/// Initializes module
/// Remark: Aborts all ongoing transfers immediately
METHOD M_Init : BOOL
VAR_INPUT
END_VAR
eHandOverState := E_HandOverState.IDLE;
DeleteNextTransportData := FALSE;
RequestNextTransportData := FALSE;
HandoverComplete := FALSE;
FastSpeed := FALSE;

M_Init := TRUE;
END_METHOD

END_FUNCTION_BLOCK

// ---- 20_Product/10_BCF/11_Conv/12_E_Functions/10_Helper/FB_HandoverTracking.TcPOU

///Handover tracking while handing over the TU from the base tracking to next function
FUNCTION_BLOCK FB_HandoverTracking IMPLEMENTS I_HandoverListener
(**************************************************************************************
* Application : BoxControl Framework 
* Revision date : $Date: 2021-03-03 11:30:54 +0100 (ons, 03 mar 2021) $
* Author : CDC
* ------------------------------------------------------------------------------------ 
* © Swisslog AG 
* Swisslog is not liable for any usage of this source code that is not agreed 
* on between Swisslog and the other party. The mandatory legal liability remains 
* unaffected. 
* ------------------------------------------------------------------------------------ 
* Project revision history: 
* 
* 	VERSION 		DATE 			INITIALS 			DESCRIPTION 
* 	0.1 			22.08.2018 		herzig 				First implementation
*	0.2				05.10.2018		b7bolm				Review
* 
**************************************************************************************)
VAR_INPUT
	Param 						: ST_TransportControlParam; // Parameter of the transport control
	NextTransportData			: ST_TransportData; // Next transport data
	Enable						: BOOL; // Transport enable
	EnableHandOver 				: BOOL; // Transport enable handover
	OccupiedSensor				: BOOL; // Occupied PE, only to detect UFOs and data missmatch
	ZoneEndLength				: UINT; // Occupied position, distance from occupied to zone end
	TrackingLength				: UDINT; // Length of tracked distance
	MaxFrontEdgeDeviation		: UDINT := 100; // Max allowed deviation between occupied sensor and allocated zone
	DisableTU_Synchronisation	: BOOL; // Disable synchronisation of TU at occupied sensor
	DriveReady					: BOOL; // Drive is ready to be used
	DriveRunning				: BOOL; // Feedback drive is running
	EncoderValueInc				: UDINT; // Encoder value [inc]
	MaxEncoderValueInc			: UDINT; // Max encoder value [inc]
	RateIncPerMM				: LREAL; // Resolution number of increments for one mm
	iWindowTracking				: I_WindowTracking;  // Window tracking implementation
END_VAR
VAR_OUTPUT
	DriveRun					: BOOL; // Drive run
	DriveStop					: BOOL; // Stop drive
	FastSpeed					: BOOL; // Fast speed possible
	RequestNextTransportData 	: BOOL; // Request next transport data
	DeleteNextTransportData  	: BOOL; // Delete next transport data
	eHandOverState				: E_HandOverState; // Handover state
	eNextTakeOverState			: E_TakeOverState; // Takeover state of next position
	Initialized					: BOOL; // Module is initialized
	HandoverOngoing				: BOOL; // Handover ongoing, interface in interaction
	HandingOverTU				: BOOL; // Handing over the TU
END_VAR
VAR_IN_OUT
	ZoneData					: ST_ZoneData; // Zone data
	ErrorData 					: ST_ErrorDataSet; // Error data
END_VAR
VAR
	fbDebugMsg					: FB_DebugMsg; // Debug instance
	DebugMsg					: T_MAXSTRING; // Debug message
	TransportComplete			: BOOL; // Transport completed
	eTrackingState 				: E_HandoverTrackingState; // Handover state machine
	fbHandover					: FB_Handover; // Basic handover impementation
	TU_StartPosition			: UDINT; // TU start position
	TU_EndPosition				: UDINT; // TU end position
	TU_DetectedOnTracking 		: BOOL; // TU detected on tracking
	EndLengthEmpty 				: BOOL; // No TU in end length found
	TrackingZoneIndex 			: UINT; // Window tracking zone index
	TrackingUfoZoneIndex 		: UINT; // Window tracking zone index of ufo
	TrackingUfoReZoneIndex 		: UINT; // Window tracking zone index of ufo rear edge
	OccupiedZoneIndex 			: UINT; // Occupied zone index
	OccupiedTracking 			: BOOL; // Occupied tracking
	TransportEnable				: BOOL; // Transport hardstop
	TransportEnableHandOver		: BOOL; // Transport softstop, finish ongoing operations
	MonitorStoppingTU_Active	: BOOL; // Monitoring state is processed currently
	fbTrigOccupied				: R_TRIG; // Only check physical and tracking distance once
	fbZoneEndLengthClear		: FB_DisplacementMeter; // ZoneEndLenght clear
	DelayLength					: UDINT; // Delay length to clear conveyor end
	ZoneEndPosition				: UDINT; // End position of zone
END_VAR

//Input mapping
TransportEnable := Enable AND Param.rZoneEnable.Transport;
TransportEnableHandOver := EnableHandOver AND Param.rZoneEnable.HandOver AND Param.rExternalZoneEnable;

F_ResetError(Reset := FALSE, ErrorData := ErrorData);	

IF iWindowTracking = 0 OR
   TrackingLength = 0 THEN
	RETURN;
END_IF

// Initialization of the module
// Module initialization
IF NOT Initialized THEN
	RETURN;
END_IF

(**************************************************************************************************************
   Synchronization / Managing of physical TUs
***************************************************************************************************************)
// Always when a TU gets detected at sensor its checked if its synchronized to tracking.
// 1. If a TU gets detected and a corresponding tracked zone is found -> Everything fine
// 2. A TU gets detected without a tracked zone, try to find corresponding zone and align
// 3. TU can not be linked to a zone, add TU as new unknown zone to the tracking

// Remark: It is possible, that there is a small difference between zone and TU when the TU leaves
// the occupied sensor. 
IF NOT DisableTU_Synchronisation THEN
	fbTrigOccupied(CLK := OccupiedSensor);
	
	IF fbTrigOccupied.Q THEN
		OccupiedTracking := iWindowTracking.M_IsTU_Present(TrackingLength - ZoneEndLength);
	
		IF OccupiedTracking THEN
			// Sensor signal is corresponding to tracking zones
			;
		ELSE
			// Try to synchronize zone to occupied signal
			OccupiedZoneIndex := iWindowTracking.M_ResyncTU_FE(
									mAbsolutePosition 		:= TrackingLength - ZoneEndLength,
									mMaxFrontEdgeDeviation 	:= MaxFrontEdgeDeviation);
		
			// If physical TU could not be linked to a zone, handle as unidentified TU
			// Add it to tracking to follow normal handover procedure
			IF OccupiedZoneIndex = 0 THEN
				TrackingUfoZoneIndex := iWindowTracking.M_AddTU_FE(
											mTU_Index 			:= 0,
											mAbsolutePosition 	:= TrackingLength - ZoneEndLength,
											miActionListener 	:= 0);
											
				fbDebugMsg.M_SendInfoMsg(CONCAT('UFO front edge detected. Created ZoneIndex: ', UINT_TO_STRING(TrackingUfoZoneIndex)));	
			END_IF
		END_IF
		
	// Ufo found, wait for rear edge	
	ELSIF TrackingUfoZoneIndex > 0 AND NOT OccupiedSensor THEN
		TrackingUfoReZoneIndex := iWindowTracking.M_AddTU_RE(
									mAbsolutePosition 	:= TrackingLength - ZoneEndLength,
									mZoneIndex 			:= TrackingUfoZoneIndex);
									
		fbDebugMsg.M_SendInfoMsg(CONCAT('UFO rear edge detected. Completed ZoneIndex: ', UINT_TO_STRING(TrackingUfoReZoneIndex)));								
		TrackingUfoZoneIndex := 0;
	END_IF
END_IF

(**************************************************************************************************************
   Tracking state
***************************************************************************************************************)
MonitorStoppingTU_Active := FALSE;

CASE eTrackingState OF
	// Idle - Wait for a TU to handover
	E_HandoverTrackingState.WAITING_FOR_TU:	
		TrackingZoneIndex := 0;
		TransportComplete := FALSE;
		ZoneData.TransportControlData.TU_DataIndex := 0;
		ZoneData.TransportControlData.DataPresent := ZoneData.TransportControlData.TU_DataIndex > 0;
		
		// Check for a TU at occupation position (REMARK: Tracking zone begin != TU begin)
		TU_DetectedOnTracking := iWindowTracking.M_IsTU_Present(TrackingLength - ZoneEndLength);
 		
		// Scan for zones between occupation point and tracking end
		IF NOT EndLengthEmpty THEN	
			TrackingZoneIndex := iWindowTracking.M_GetLastZoneIndex(TrackingLength - ZoneEndLength , TrackingLength, TRUE);
			
			// A zone with TU present was found
			IF TrackingZoneIndex > 0 THEN
				// Get rear edge position of TU
				TU_EndPosition := iWindowTracking.M_GetTU_EndPosition(TrackingZoneIndex);
				// Check if TU already left conveyor
				IF TU_EndPosition > TrackingLength THEN
					// Get end position of zone
					ZoneEndPosition := iWindowTracking.M_GetZoneEndPosition(TrackingZoneIndex);
					
					// Search 2nd last zone, since TU of last zone already left conveyor
					IF ZoneEndPosition > (TrackingLength - ZoneEndLength) THEN
						TrackingZoneIndex := iWindowTracking.M_GetLastZoneIndex(TrackingLength - ZoneEndLength , ZoneEndPosition - 1, TRUE);
					ELSE
						// No zone found
						TrackingZoneIndex := 0;
					END_IF
				END_IF
				
				// A zone with a TU which is still on conveyor was found
				IF TrackingZoneIndex > 0 THEN 
					ZoneData.TransportControlData.TU_DataIndex := iWindowTracking.P_ZoneTable[TrackingZoneIndex].TU_Index;
					ZoneData.TransportControlData.DataPresent := ZoneData.TransportControlData.TU_DataIndex > 0;
					eTrackingState := E_HandoverTrackingState.MONITOR_STOPPING_TU;
				ELSE
					EndLengthEmpty := TRUE;
				END_IF
			ELSE
				EndLengthEmpty := TRUE;
			END_IF
			
		ELSIF TU_DetectedOnTracking  THEN
			// Get corresponding zone index
			TrackingZoneIndex := iWindowTracking.M_GetZoneIndex(TrackingLength - ZoneEndLength);
			EndLengthEmpty := FALSE;
			
			IF TrackingZoneIndex > 0 THEN
				ZoneData.TransportControlData.TU_DataIndex := iWindowTracking.P_ZoneTable[TrackingZoneIndex].TU_Index;
				ZoneData.TransportControlData.DataPresent := ZoneData.TransportControlData.TU_DataIndex > 0;
			END_IF
			
			eTrackingState := E_HandoverTrackingState.MONITOR_STOPPING_TU;
		END_IF
	
	// Handover is not initiated, ensure TU can stop properly
	E_HandoverTrackingState.MONITOR_STOPPING_TU:
		MonitorStoppingTU_Active := TRUE;
	
		IF TrackingZoneIndex > 0 THEN
			TU_StartPosition := iWindowTracking.M_GetTU_StartPosition(TrackingZoneIndex);
			
			// When zone is not in a valid range, forget index (> Occupation point)
			IF TU_StartPosition < (TrackingLength - ZoneEndLength) OR 
               NOT iWindowTracking.P_ZoneTable[TrackingZoneIndex].Used THEN
				TrackingZoneIndex := 0;
				DriveStop := FALSE;
				
				MonitorStoppingTU_Active := FALSE;
				eTrackingState := E_HandoverTrackingState.WAITING_FOR_TU;
				RETURN;
				
			// Check for overrun
			ELSIF TU_StartPosition > TrackingLength AND 
               iWindowTracking.P_ZoneTable[TrackingZoneIndex].TU_Index > 0 THEN
				// Overrun detected - Handover was not initated and TU could not stop on Tracking
				// Maybe condition to stop is wrong or available breaking distance is to short
				// Possible TU Index get deleted, because a crash could happen what maybe leads to 
				// Tu data inconsistency.
				iWindowTracking.P_ZoneTable[TrackingZoneIndex].TU_Index := 0;
				ZoneData.TransportControlData.TU_DataIndex := 0;
				ZoneData.TransportControlData.DataPresent := ZoneData.TransportControlData.TU_DataIndex > 0;
				fbDebugMsg.M_SendInfoMsg(CONCAT('Handover not initiated, TU_DataIndex deleted. ZoneIndex: ', UINT_TO_STRING(TrackingZoneIndex)));	
			END_IF
			
			// Wait until handover is initiated resp. ongoing
			IF fbHandover.eHandOverState = E_HandOverState.ACTIVE OR
			   fbHandover.eHandOverState = E_HandOverState.STOP OR
			   fbHandover.eHandOverState = E_HandOverState.INTERRUPTED OR 
               eNextTakeoverState = E_TakeOverState.ACTIVE THEN
			   
			   MonitorStoppingTU_Active := FALSE;
			   eTrackingState := E_HandoverTrackingState.MONITOR_HANDOVER_TU;
			END_IF
		ELSE
			MonitorStoppingTU_Active := FALSE;
			eTrackingState := E_HandoverTrackingState.WAITING_FOR_TU;
		END_IF
	
	// Handover was initiated, wait until TU left position
	E_HandoverTrackingState.MONITOR_HANDOVER_TU:
		IF TrackingZoneIndex > 0 THEN
			TU_StartPosition := iWindowTracking.M_GetTU_StartPosition(TrackingZoneIndex);
			TU_EndPosition := iWindowTracking.M_GetTU_EndPosition(TrackingZoneIndex);
			
			// Monitor zone if it is not in a valid range, forget index (> Occupation point)
			IF TU_StartPosition < (TrackingLength - ZoneEndLength) OR 
			   NOT iWindowTracking.P_ZoneTable[TrackingZoneIndex].Used THEN
				TrackingZoneIndex := 0;
				eTrackingState := E_HandoverTrackingState.WAITING_FOR_TU;
				RETURN;

			// Wait until transport is completed by
			// - Zone not available anymore
			// - Not occupied anymore
			// - Transport aborted or completed
			ELSIF NOT iWindowTracking.P_ZoneTable[TrackingZoneIndex].Used OR
			      NOT iWindowTracking.P_ZoneTable[TrackingZoneIndex].TU_Present OR
 			      fbHandover.eHandOverState = E_HandOverState.IDLE OR 
			      fbHandover.eHandOverState = E_HandOverState.UNDEFINED OR 
                  TransportComplete THEN		
				eTrackingState := E_HandoverTrackingState.WAITING_FOR_TU;
				
			// Monitor TU-DataIndex, and update it when it was deleted during handover
			ELSIF ZoneData.TransportControlData.TU_DataIndex <> iWindowTracking.P_ZoneTable[TrackingZoneIndex].TU_Index THEN
				iWindowTracking.P_ZoneTable[TrackingZoneIndex].TU_Index := ZoneData.TransportControlData.TU_DataIndex;
			END_IF
		ELSE
			eTrackingState := E_HandoverTrackingState.WAITING_FOR_TU;
		END_IF
// Default
ELSE
	eTrackingState := E_HandoverTrackingState.WAITING_FOR_TU;
END_CASE

(**************************************************************************************************************
   Handover state
***************************************************************************************************************)
// If an index was found between occupation point and tracking length
// Wait until TU left occupation point, to zone end length for handover
IF TrackingZoneIndex > 0 THEN 
	IF NOT fbZoneEndLengthClear.Run THEN
		TU_EndPosition := iWindowTracking.M_GetTU_EndPosition(TrackingZoneIndex);
		// TU rear edge is between occupied point and conveyor end
		IF (TrackingLength - ZoneEndLength) < TU_EndPosition AND TrackingLength >= TU_EndPosition THEN
			// Calculate distance from  TU rear edge to conveyor end 
			DelayLength := TrackingLength - TU_EndPosition;
		
			// Run zone end length clearing 
			fbZoneEndLengthClear(
				Run 				:= fbHandover.HandoverOngoing, 
				EncoderValueInc		:= EncoderValueInc,
				MaxEncoderValueInc 	:= MaxEncoderValueInc,
				RateIncPerMM		:= RateIncPerMM,
				SetPoint 			:= UDINT_TO_UINT(DelayLength));
		END_IF
	END_IF
END_IF

fbZoneEndLengthClear(
	EncoderValueInc		:= EncoderValueInc,
	MaxEncoderValueInc 	:= MaxEncoderValueInc,
	RateIncPerMM		:= RateIncPerMM);
	
fbHandover(
	Enable					:= TransportEnable AND
            				  (Param.rOperationState.eState = E_PositionState.STARTED OR
	        				   Param.rOperationState.eState = E_PositionState.STOPPING),
	RequestHandover			:= TrackingZoneIndex > 0 AND Param.rOperationState.eState = E_PositionState.STARTED AND TransportEnableHandOver,
	NextZonePresent			:= Param.reNextFunctionNumber > 0,
	HandoverComplete		:= fbZoneEndLengthClear.Q,
	DriveReady				:= DriveReady,
	iListener				:= THIS^,
	FastSpeed				=> FastSpeed,
	DriveRun				=> DriveRun,
	eHandOverState			=> eHandOverState,
	eNextTakeOverState		=> eNextTakeOverState,
	RequestNextTransportData=> RequestNextTransportData,
	DeleteNextTransportData	=> DeleteNextTransportData,
	HandoverOngoing			=> HandoverOngoing,
	NextTransportData		:= NextTransportData,
	ErrorData				:= ErrorData);

IF fbZoneEndLengthClear.Q THEN
	fbZoneEndLengthClear(RUN := FALSE);
END_IF

ZoneData.TransportControlData.eHandOverState := eHandOverState;
ZoneData.TransportControlData.DataPresent := ZoneData.TransportControlData.TU_DataIndex <> 0;
ZoneData.TransportControlData.SensorOccupied := iWindowTracking.M_IsTU_Present(TrackingLength - ZoneEndLength);
ZoneData.TransportControlData.TU_LeadingEdgePos := 0;

DriveStop := (fbHandover.HandoverOngoing AND NOT fbHandover.DriveRun AND NOT fbHandover.DriveRequest) OR 
             (NOT fbHandover.HandoverOngoing AND MonitorStoppingTU_Active AND
			  (eHandOverState <> E_HandoverState.READY OR eNextTakeOverState <> E_TakeOverState.READY));

HandingOverTU := fbHandOver.HandoverOngoing;

/// Handover completed event
METHOD M_HandoverCompleteEvent

IF eTrackingState = E_HandoverTrackingState.MONITOR_HANDOVER_TU THEN
	TransportComplete := TRUE;
	
	IF iWindowTracking <> 0 THEN
		IF TrackingZoneIndex > 0 THEN
			iWindowTracking.M_DeleteZone(mZoneIndex := TrackingZoneIndex);
		END_IF
	END_IF
END_IF
END_METHOD

METHOD M_HandoverStartEvent
END_METHOD

/// Initialize module
METHOD M_Init : BOOL
VAR_INPUT
END_VAR
fbHandover.M_Init();

eTrackingState := E_HandoverTrackingState.WAITING_FOR_TU;
Initialized := TRUE;
M_Init := TRUE;
END_METHOD

END_FUNCTION_BLOCK

// ---- 20_Product/30_Toolbox/17_WindowTracking/10_Core/FB_DisplacementMeter.TcPOU
FUNCTION_BLOCK FB_DisplacementMeter
(**************************************************************************************
 * 	Application		:	BoxControl Framework
 *	Revision		:	$Revision: 354283 $
 *	Revision date	:	$Date: 2015-09-02 11:51:42 +0200 (Mi, 02 Sep 2015) $
 *	Last changed by	:	$Author: d7mangc $
 *	URL				:	$URL: http://almscdc.swisslog.com/repo/SWPD/Development/BoxControlFramework/20_Release/trunk/01_Software/BoxControlFramework/BoxControlFramework/JumpStart/11_Library/10_Application/10_Base/13_TimerCounter/FB_Timer.TcPOU $
 *
 *	Purpose			:	Measures displacement based on encoder value. Output Q gets true when setpoint is reached
 *						
 *
 * ------------------------------------------------------------------------------------
 *	Copyright Swisslog [IP AG], Switzerland. All rights reserved.
 * 
 * ------------------------------------------------------------------------------------
 *	
 * 	Revision History: 
 *
 * 	VERSION			DATE			INITIALS			DESCRIPTION
 *	0.1				01.01.2001		swl					Example
 *
 **************************************************************************************)
VAR_INPUT
	Run             	: BOOL; // Start process on rising edge
	EncoderValueInc		: UDINT; // Encoder value [inc], Ascending = forward
	MaxEncoderValueInc	: UDINT; // Max encoder value [inc]
	RateIncPerMM		: LREAL; // Ratio - How many increments represent one mm
	SetPoint			: DINT; // Displacement value where Q is set true (negative: backward direction, positive: forward direction)
	StartPoint		    : DINT; // Starting position (offset) for displacement measurement [mm] (negative : backward direction, positive: forward direction)
END_VAR
VAR_OUTPUT
	Q		 			: BOOL; // True when setpoint reached
	DisplacementInc		: DINT; // Current displacement [inc] (negative : backward direction, positive: forward direction)
	Displacement		: DINT; // Current displacement [mm] (negative : backward direction, positive: forward direction)
END_VAR
VAR
	Trg			     	: BOOL; // Trigger detection for start signal
	LastEncoderValueInc	: UDINT; // Last encoder value [inc]
	Inc 			 	: DINT; // increments
END_VAR

IF Run THEN
	// Detect start trigger and preset values
	IF NOT Trg AND Run THEN
		LastEncoderValueInc := EncoderValueInc;
		DisplacementInc := LREAL_TO_DINT(DINT_TO_LREAL(StartPoint) * RateIncPerMM);
		Displacement := 0;
	END_IF

	Inc := UDINT_TO_DINT(EncoderValueInc) - UDINT_TO_DINT(LastEncoderValueInc);
	IF ABS(Inc) > UDINT_TO_DINT(MaxEncoderValueInc/2) THEN
		IF Inc < 0 THEN
			Inc := Inc + 1 + UDINT_TO_DINT(MaxEncoderValueInc);
		ELSE
			Inc := UDINT_TO_DINT(EncoderValueInc) - (UDINT_TO_DINT(LastEncoderValueInc) + UDINT_TO_DINT(MaxEncoderValueInc)) - 1;
		END_IF
	END_IF
	
	// Update last encoder value
	LastEncoderValueInc := EncoderValueInc;
	
	// Update outputs
	IF NOT Q THEN
		DisplacementInc := DisplacementInc + Inc;
		
		IF RateIncPerMM > 0 THEN
			Displacement := LREAL_TO_DINT(DINT_TO_LREAL(DisplacementInc) / RateIncPerMM);
		ELSE
			Displacement := 0;
		END_IF
		
		// To ensure counting direction is as desired,
		// decision is based on the sign of setpoint
		IF SetPoint >= 0 THEN
			IF Displacement >= SetPoint THEN
				Q := TRUE;
			END_IF
		ELSE
			IF Displacement <= SetPoint THEN
				Q := TRUE;
			END_IF
		END_IF
	END_IF
ELSE
	// Reset outputs
	Q := FALSE;
END_IF

Trg := Run;

END_FUNCTION_BLOCK

// ---- 20_Product/10_BCF/11_Conv/12_E_Functions/10_Helper/FB_HandoverTrackingDivert.TcPOU
/// Functionality to control a handover process from a tracking conveyor
FUNCTION_BLOCK FB_HandoverTrackingDivert IMPLEMENTS I_HandoverListener
(************************************************************************************** 
* 	Application 		: BoxControl Framework 
* 	Revision 			: $Revision: 408723 $ 
* 	Revision date 		: $Date: 2018-06-27 13:49:08 +0200 (Wed, 27 Jun 2018) $ 
* 	Last changed by 	: $Author: b7bolm $ 
* 	URL 				: $URL: http://almscdc.swisslog.com/repo/SWPD/Development/BoxControlFramework/21_Projects/BCF_2.0/trunk/BCF/BCF/JumpStart/20_Product/10_App/12_E_Functions/10_Lib/10_Conv/FB_FunctionList.TcPOU $ 
* ------------------------------------------------------------------------------------ 
* 	© Swisslog AG 
* 	Swisslog is not liable for any usage of this source code that is not agreed 
* 	on between Swisslog and the other party. The mandatory legal liability remains 
* 	unaffected. 
* ------------------------------------------------------------------------------------ 
* 	Revision History: 
* 
* 	VERSION 		DATE 			INITIALS 			DESCRIPTION 
* 	0.1 			22.08.2018 		herzig 				First implementation
*	0.2				05.10.2018		b7bolm				Review
* 
**************************************************************************************)
VAR_INPUT
	Param 						: ST_TransportControlParam; // Parameter of the transport control
	NextTransportData			: ST_TransportData; // Next transport data
	Enable						: BOOL; // Transport enable
	EnableHandOver 				: BOOL; // Transport enable handover
	DivertPosition				: UDINT; // Merging position on tracking
	DivertingTolerance			: UDINT; // Merging tolerance to allow merging
	DivertRearEdge				: BOOL; // Divert on rear edge of TU
	DriveDelayDistance			: DINT;  // Distance to drive until position is free
	DriveReady					: BOOL; // Drive is ready to be used
	EncoderValueInc				: UDINT; // Encoder value [inc]
	MaxEncoderValueInc			: UDINT; // Max encoder value [inc]
	RateIncPerMM				: LREAL; // Resolution amount of increment per mm
	iWindowTracking				: I_WindowTracking;  // Window tracking implementation
END_VAR

VAR_OUTPUT
	DriveRun					: BOOL; // Drive run
	DriveStop					: BOOL; // Stop drive
	FastSpeed					: BOOL; // Fast speed possible
	RequestNextTransportData 	: BOOL; // Request next transport data
	DeleteNextTransportData  	: BOOL; // Delete next transport data
	eHandOverState				: E_HandOverState; // Handover state
	eNextTakeOverState			: E_TakeOverState; // Takeover state of next position
	Initialized					: BOOL; // Module is initialized
	AvailableZoneIndex			: UINT; // Current valid zone index
	HandoverOngoing				: BOOL; // Handover ongoing, interface in interaction
END_VAR

VAR_IN_OUT
	ZoneData					: ST_ZoneData; // Zone data
	ErrorData 					: ST_ErrorDataSet; // Error data
END_VAR

VAR
	fbDebugMsg					: FB_DebugMsg; // Debug instance
	DebugMsg					: T_MAXSTRING; // Debug message
	fbHandover					: FB_Handover; // Basic handover impementation
	DistanceToTU				: DINT; // Distance to TU from diverting point
	TransportEnable				: BOOL; // Transport hardstop
	TransportEnableHandOver		: BOOL; // Transport softstop, finish ongoing operations
	TU_IndexOfZone				: DINT; // TU index of tracking zone
	TrackingZoneIndex 			: UINT; // Tracking zone index
	fbZoneEndLengthClear		: FB_DisplacementMeter; // ZoneEndLenght clear
END_VAR

//Input mapping
TransportEnable := Enable AND Param.rZoneEnable.Transport;
TransportEnableHandOver := EnableHandOver AND Param.rZoneEnable.HandOver AND Param.rExternalZoneEnable;

F_ResetError(Reset := FALSE, ErrorData := ErrorData);	

IF iWindowTracking = 0 THEN
	RETURN;
END_IF

// Initialization of the module
// Module initialization
IF NOT Initialized THEN
	RETURN;
END_IF

(**************************************************************************************************************
   Determine zone for this position
***************************************************************************************************************)
AvailableZoneIndex := 0;
TU_IndexOfZone := 0;
ZoneData.TransportControlData.DataPresent := FALSE;
ZoneData.TransportControlData.TU_DataIndex := 0;

// Wait until a zone can be found at divert point
IF TrackingZoneIndex = 0 THEN
	IF DivertRearEdge THEN
		TrackingZoneIndex := iWindowTracking.M_GetFirstZoneIndex(DivertPosition, DivertPosition + DivertingTolerance, TRUE);
	ELSE
		TrackingZoneIndex := iWindowTracking.M_GetZoneIndex(DivertPosition);	
	END_IF
END_IF

// When a possible zone was found, validate and monitor it
IF TrackingZoneIndex > 0 THEN
	// As long the zone is valid
	IF iWindowTracking.P_ZoneTable[TrackingZoneIndex].Used THEN
		// Divert on rear edge
		IF DivertRearEdge THEN
			// Zone gets monitored as long it is in a certain range 
			DistanceToTU := iWindowTracking.M_GetDistanceToTU_End(DivertPosition, TrackingZoneIndex);
		ELSE
			// Zone gets monitored as long it is in a certain range 
			DistanceToTU := iWindowTracking.M_GetDistanceToTU_Start(DivertPosition, TrackingZoneIndex);
		END_IF
		
		// TU needs to pass divert point and stays available for distance (Divertingtolerance)
		IF DistanceToTU <= 0 AND ABS(DistanceToTU) <= UDINT_TO_DINT(DivertingTolerance) THEN
			// When position is occupied, its a possible next for this position
			IF iWindowTracking.P_ZoneTable[TrackingZoneIndex].TU_Present THEN			
				TU_IndexOfZone := iWindowTracking.P_ZoneTable[TrackingZoneIndex].TU_Index;
			
				ZoneData.TransportControlData.DataPresent := TU_IndexOfZone <> 0;
				ZoneData.TransportControlData.TU_DataIndex := TU_IndexOfZone;
				
				AvailableZoneIndex := TrackingZoneIndex;	
			END_IF
			
		// TU left divert tolerance range
		ELSIF DistanceToTU <= 0 AND ABS(DistanceToTU) > UDINT_TO_DINT(DivertingTolerance) THEN
			TrackingZoneIndex := 0;
		END_IF
	END_IF
END_IF

(**************************************************************************************************************
   Handover state
***************************************************************************************************************)
// Delay after enabling handover, set as soon transport gets started
fbZoneEndLengthClear(
	EncoderValueInc		:= EncoderValueInc,
	MaxEncoderValueInc 	:= MaxEncoderValueInc,
	RateIncPerMM		:= RateIncPerMM);
	
fbHandover(
	Enable					:= TransportEnable AND
            				  (Param.rOperationState.eState = E_PositionState.STARTED OR
	         				   Param.rOperationState.eState = E_PositionState.STOPPING),
	RequestHandover			:= AvailableZoneIndex > 0 AND Param.rOperationState.eState = E_PositionState.STARTED AND TransportEnableHandOver,
	NextZonePresent			:= Param.reNextFunctionNumber > 0,
	HandoverComplete		:= fbZoneEndLengthClear.Q,
	DriveReady				:= DriveReady,
	iListener				:= THIS^,
	FastSpeed				=> FastSpeed,
	DriveRun				=> DriveRun,
	eHandOverState			=> eHandOverState,
	eNextTakeOverState		=> eNextTakeOverState,
	RequestNextTransportData=> RequestNextTransportData,
	DeleteNextTransportData	=> DeleteNextTransportData,
	HandoverOngoing			=> HandoverOngoing,
	NextTransportData		:= NextTransportData,
	ErrorData				:= ErrorData);
	
IF fbZoneEndLengthClear.Q THEN
	fbZoneEndLengthClear(RUN := FALSE);
END_IF
	
ZoneData.TransportControlData.eHandOverState := eHandOverState;
ZoneData.TransportControlData.DataPresent := ZoneData.TransportControlData.TU_DataIndex <> 0;
ZoneData.TransportControlData.SensorOccupied := AvailableZoneIndex > 0;
ZoneData.TransportControlData.Occupied := AvailableZoneIndex > 0;
ZoneData.TransportControlData.TU_LeadingEdgePos := 0;

DriveStop := (fbHandover.HandoverOngoing AND NOT fbHandover.DriveRun AND NOT fbHandover.DriveRequest);

/// Handover completed event
METHOD M_HandoverCompleteEvent
TrackingZoneIndex := 0;
END_METHOD

/// Handover initiated -> Active
METHOD M_HandoverStartEvent
VAR
	mZoneDeleted	: BOOL;
END_VAR

IF AvailableZoneIndex > 0 THEN
	IF iWindowTracking <> 0 THEN
		mZoneDeleted := iWindowTracking.M_DeleteZone(AvailableZoneIndex);
		IF mZoneDeleted THEN
			DebugMsg := CONCAT('Zone deleted from tracking by divert. ZoneIndex: ', UINT_TO_STRING(AvailableZoneIndex));
			
		ELSE
			DebugMsg := CONCAT('Zone delete from tracking by divert not possible. ZoneIndex: ', UINT_TO_STRING(AvailableZoneIndex));
		END_IF
		fbDebugMsg.M_SendInfoMsg(DebugMsg);
	END_IF
	
	// Run zone end length clearing 
	fbZoneEndLengthClear(
		Run 				:= TRUE, 
		EncoderValueInc		:= EncoderValueInc,
		MaxEncoderValueInc 	:= MaxEncoderValueInc,
		RateIncPerMM 		:= RateIncPerMM,
		SetPoint 			:= DriveDelayDistance);
END_IF
END_METHOD

/// Initialize module
METHOD M_Init : BOOL
VAR_INPUT
END_VAR
fbHandover.M_Init();

Initialized := TRUE;
M_Init := TRUE;
END_METHOD

END_FUNCTION_BLOCK

// ---- 20_Product/10_BCF/11_Conv/12_E_Functions/10_Helper/FB_SpeedControl.TcPOU
FUNCTION_BLOCK FB_SpeedControl
(**************************************************************************************
 * 	Application		:	BoxControl Framework
 *	Revision		:	$Revision: 404529 $
 *	Revision date	:	$Date: 2018-04-23 08:21:38 +0200 (Mo., 23 Apr 2018) $
 *	Last changed by	:	$Author: b7bolm $
 *	URL				:	$URL: http://almscdc.swisslog.com/repo/SWPD/Development/BoxControlFramework/20_Release/trunk/01_Software/BCF/BCF/JumpStart/20_Product/10_App/12_E_Functions/10_Lib/10_Conv/10_Functions/FB_SpeedControl.TcPOU $
 *
 *	Purpose			:	Speed control
 *
 * ------------------------------------------------------------------------------------
 *	Copyright Swisslog [IP AG], Switzerland. All rights reserved.
 * 
 * ------------------------------------------------------------------------------------
 *	
 * 	Revision History: 
 *
 * 	VERSION			DATE			INITIALS			DESCRIPTION
 *	0.1				01.01.2001		swl					Example
 *
 **************************************************************************************)
VAR_INPUT
	FastSpeed 		: BOOL; // Fast speed
	SetSpeed 		: REAL; // Set speed of the zone [m/s]
	SpeedSlow 		: INT;  // Speed slow [%]
	SpeedFast 		: INT;  // Speed fast [%]
END_VAR

VAR
	MasterSpeed		: INT; // Master speed [%]
END_VAR

VAR_OUTPUT
	CommandSpeed 	: INT; // Command speed [mm/s]
END_VAR

// Get Master speed from subsystem
IF __ISVALIDREF(SubsystemRegistry.rSubsystemInterface) THEN
	MasterSpeed := SubsystemRegistry.rSubsystemInterface.Out.MasterSpeed;
ELSE
	MasterSpeed := 100;
END_IF

// Calculate command speed
IF FastSpeed THEN
	CommandSpeed := REAL_TO_INT(SetSpeed * 1000 * SpeedFast / 100 * MasterSpeed / 100);
ELSE
	CommandSpeed := REAL_TO_INT(SetSpeed * 1000 * SpeedSlow / 100 * MasterSpeed / 100);
END_IF

END_FUNCTION_BLOCK

// ---- 20_Product/10_BCF/11_Conv/12_E_Functions/10_Helper/FB_SpeedControlRamp.TcPOU
FUNCTION_BLOCK FB_SpeedControlRamp
(**************************************************************************************
 * 	Application		:	BoxControl Framework
 *	Revision		:	$Revision: 404529 $
 *	Revision date	:	$Date: 2018-04-23 08:21:38 +0200 (Mo., 23 Apr 2018) $
 *	Last changed by	:	$Author: b7bolm $
 *	URL				:	$URL: http://almscdc.swisslog.com/repo/SWPD/Development/BoxControlFramework/20_Release/trunk/01_Software/BCF/BCF/JumpStart/20_Product/10_App/12_E_Functions/10_Lib/10_Conv/10_Functions/FB_SpeedControl.TcPOU $
 *
 *	Purpose			:	Speed control with acceleration/deceleration ramps
 *
 * ------------------------------------------------------------------------------------
 *	Copyright Swisslog [IP AG], Switzerland. All rights reserved.
 * 
 * ------------------------------------------------------------------------------------
 *	
 * 	Revision History: 
 *
 * 	VERSION			DATE			INITIALS			DESCRIPTION
 *	0.1				01.01.2001		swl					Example
 *
 **************************************************************************************)
VAR_INPUT
	DriveRun 				: BOOL; // Drive run
	TU_InBrakingZone 		: BOOL; // TU is within the braking zone 
	SetSpeed 				: REAL; // Set speed of the zone [m/s]
	SpeedSlow 				: INT; // Speed slow [%]
	SpeedFast 				: INT; // Speed fast [%]
	Acceleration   	 		: INT; // Accelaration [mm/s^2]
	Deceleration   	 		: INT; // Deceleration [mm/s^2]
	TransportControlData 	: ST_TransportControlData;
	SpeedPrevZone			: INT; // Speed from previous zone
	MinimumSpeed			: INT; // Minimum speed [mm/s]
END_VAR
VAR
	MasterSpeed				: INT; // Master speed [%]
	fbGetCurTaskIdx  		: GETCURTASKINDEX;
	CycleTime       		: REAL; // System cycletime [s]
	DesiredSpeed 			: INT; // Desired speed [mm/s]
	State 					: E_SpeedControlState; // Speed control state
	SpeedDelta				: INT; // Speed delta [mm/s]
END_VAR
VAR_OUTPUT
	CommandSpeed 			: INT; // Command speed [mm/s]
END_VAR

// Get current cycle time
fbGetCurTaskIdx();
CycleTime := UDINT_TO_REAL(_TaskInfo[fbGetCurTaskIdx.index].CycleTime) / 10000000;

// Get Master speed from subsystem
IF __ISVALIDREF(SubsystemRegistry.rSubsystemInterface) THEN
	MasterSpeed := SubsystemRegistry.rSubsystemInterface.Out.MasterSpeed;
ELSE
	MasterSpeed := 100;
END_IF


(**********************************************************************************************************
   Calculate desired speed
***********************************************************************************************************)
// When TakeOver starts sync CommandSpeed with previous zone
IF TransportControlData.eTakeOverState = E_TakeOverState.READY AND
   TransportControlData.eTransportState <> E_TransportState.MULTI_TU THEN
	CommandSpeed := SpeedPrevZone;
	
// In TakeOver sync desired speed with previous zone
ELSIF TransportControlData.eTransportState = E_TransportState.TAKEOVER AND NOT TU_InBrakingZone THEN
	DesiredSpeed := SpeedPrevZone;

// Check if fast speed is active then run at fast speed	
ELSIF TransportControlData.FastSpeedActive THEN
	DesiredSpeed := REAL_TO_INT(SetSpeed * 1000 * SpeedFast / 100 * MasterSpeed / 100);
	
// When not in braking zone run at low speed
ELSIF NOT TU_InBrakingZone THEN
	DesiredSpeed := REAL_TO_INT(SetSpeed * 1000 * SpeedSlow / 100 * MasterSpeed / 100);
	
// If not in TakeOver, Fast speed and TU is in braking zone request for minimum speed
ELSE
	DesiredSpeed := MinimumSpeed;
END_IF

// Limit the desired speed between system MinimumSpeed and the zone SetSpeed
IF DriveRun THEN
	DesiredSpeed := LIMIT(MinimumSpeed, DesiredSpeed, REAL_TO_INT(SetSpeed * 1000.0));	
END_IF


(**********************************************************************************************************
   Speed control state
***********************************************************************************************************)
CASE State OF
	
// STOPPED
	E_SpeedControlState.STOPPED:
		DesiredSpeed := 0;
		CommandSpeed := 0;
		// Wait for run command  
		IF DriveRun THEN
			State := E_SpeedControlState.Accelerate;
		END_IF
		
// ACCELERATE
	E_SpeedControlState.ACCELERATE:
		IF NOT DriveRun THEN
			State := E_SpeedControlState.Stopped;
			
		ELSIF CommandSpeed >= DesiredSpeed THEN
		 	State := E_SpeedControlState.Running;
		ELSE
			// Cyclic delta in speed [mm/s / cycle]
			SpeedDelta := REAL_TO_INT(Acceleration * CycleTime);
			CommandSpeed := LIMIT(MinimumSpeed, CommandSpeed + SpeedDelta, REAL_TO_INT(SetSpeed * 1000.0));
		END_IF
		
// RUNNING	
	E_SpeedControlState.RUNNING:
		IF NOT DriveRun THEN
			State := E_SpeedControlState.Stopped;
			
		ELSIF CommandSpeed > DesiredSpeed THEN
			State := E_SpeedControlState.Decelerate;
			
		ELSIF CommandSpeed < DesiredSpeed THEN
			State := E_SpeedControlState.Accelerate;
		END_IF
	
// DECELERATE	
	E_SpeedControlState.DECELERATE:
		IF NOT DriveRun THEN
			State := E_SpeedControlState.Stopped;
			
		ELSIF CommandSpeed < DesiredSpeed THEN
			State := E_SpeedControlState.Accelerate;		
		ELSE
			// Cyclic delta in speed [mm/s / cycle]
			SpeedDelta := REAL_TO_INT(Deceleration * CycleTime);
			CommandSpeed := LIMIT(MinimumSpeed, CommandSpeed - SpeedDelta, REAL_TO_INT(SetSpeed * 1000.0));
		END_IF
	
ELSE
	State := E_SpeedControlState.STOPPED;
END_CASE

END_FUNCTION_BLOCK

// ---- 20_Product/10_BCF/11_Conv/12_E_Functions/10_Helper/FB_Takeover.TcPOU
/// Basic takeover implementation to satisfy interface
FUNCTION_BLOCK FB_Takeover
(**************************************************************************************
* Application : BoxControl Framework 
* Revision date : $Date: 2021-04-01 10:33:04 +0200 (tor, 01 apr 2021) $
* Author : CDC
* ------------------------------------------------------------------------------------ 
* © Swisslog AG 
* Swisslog is not liable for any usage of this source code that is not agreed 
* on between Swisslog and the other party. The mandatory legal liability remains 
* unaffected. 
* ------------------------------------------------------------------------------------ 
* Project revision history: 
* 
* VERSION 	DATE 		INITIALS 	DESCRIPTION 
* 	VERSION 		DATE 			INITIALS 			DESCRIPTION 
* 	0.1 			22.08.2018 		herzig 				First implementation
*	0.2				05.10.2018		b7bolm				Review
* 
**************************************************************************************)

VAR_INPUT
	Enable						: BOOL; // Allow handover in general  
	RequestTakeover				: BOOL; // Rising edge initiates a new transport
	AbortTakeover				: BOOL; // Takeover must be aborted
	PrevZonePresent 			: BOOL;	 // Previous zone is known
	EncoderValue				: UDINT; // Encoder signal of movement
	MaxEncoderValue 			: UDINT; // Maximum encoder signal
	EncoderRate					: LREAL; // Rate from encoder to mm signal
	DriveReady					: BOOL; // Drive is ready to be used
	iListener 					: I_TakeoverListener; // Listener for any takeover events
END_VAR
VAR_OUTPUT
	DriveRun					: BOOL; // Switch on drive
	DriveRequest				: BOOL; // Request to get drive ready
	eTakeOverState				: E_TakeOverState; // Takeover state
	ePrevHandOverState			: E_HandOverState; // Handoverstate of previous zone
	RequestPrevTransportData 	: BOOL; // Request previous transport data
	DeletePrevTransportData 	: BOOL; // Delete previous transport dat
	TakeoverOngoing				: BOOL; // A takeover is ongoing, statemachine in operation
END_VAR
VAR_IN_OUT
	PrevTransportData			: ST_TransportData; // Next transport data
	ErrorData					: ST_ErrorDataSet; // Error slot
END_VAR
VAR
	TU_Index					: DINT; // TU index
	fbDebugMsg					: FB_DebugMsg; // Debug instance
	DebugMsg					: T_MAXSTRING; // Debug message
END_VAR


F_ResetError(Reset := FALSE, ErrorData := ErrorData);	

(*************************************************************************
  Undefined
*************************************************************************)
CASE eTakeOverState OF
	// Undefined
	E_TakeOverState.UNDEFINED:
		TakeoverOngoing := FALSE;
		eTakeOverState := E_TakeOverState.IDLE;


(*************************************************************************
  Idle
*************************************************************************)
	E_TakeOverState.IDLE:
		TakeoverOngoing := FALSE;
		DeletePrevTransportData := FALSE;
		RequestPrevTransportData := NOT PrevZonePresent;
		DriveRequest := FALSE;
		DriveRun := FALSE;
		
		IF RequestTakeover THEN
			// If the zone is internally ready for takeover
			IF Enable  AND
			   ErrorData.ErrorType <> E_ErrorType.ERROR THEN
				  
				// If prev zone or function is available
				IF PrevZonePresent THEN
					IF PrevTransportData.rTransportControlData.eHandOverState = E_HandOverState.READY THEN
						DriveRequest := TRUE;
						
						IF DriveReady THEN
							eTakeOverState := E_TakeOverState.READY;
						END_IF
					END_IF
				END_IF
			END_IF
		END_IF


(*************************************************************************
  Ready
*************************************************************************)
	E_TakeOverState.READY:
		TakeoverOngoing := FALSE;

		IF NOT Enable OR NOT RequestTakeover OR
		   ErrorData.ErrorType = E_ErrorType.ERROR OR
           NOT PrevZonePresent OR
           NOT DriveReady THEN  
			eTakeOverState := E_TakeOverState.IDLE;

		// Previous position is ready to handover
		ELSIF PrevTransportData.rTransportControlData.eHandOverState = E_HandOverState.READY THEN
			// Set drive on to create minimum TU gap
			DriveRun := TRUE;
			
			IF iListener <> 0 THEN
			   iListener.M_TakeoverStartEvent();
		   	END_IF

			// Move TU-data index from previous to own zone
			TU_Index := F_MoveTU_DataIndex(
								eFunctionNumber := PrevTransportData.eFunctionNumber,
								mZoneNumber 	:= PrevTransportData.ZoneNumber);

			IF iListener <> 0 THEN
				iListener.M_TU_IndexMovedEvent(TU_Index);
			END_IF

			eTakeOverState := E_TakeOverState.ACTIVE;
		END_IF


(*************************************************************************
  Active
*************************************************************************)
	E_TakeOverState.ACTIVE:
		DriveRun := TRUE;
		DriveRequest := FALSE;
		
		// Interrupt takeover if previous position stopped handover
		IF PrevTransportData.rTransportControlData.eHandOverState = E_HandOverState.STOP THEN
			DriveRun := FALSE;
			eTakeOverState := E_TakeOverState.INTERRUPTED;

		// Stop takeover from own cause
		ELSIF NOT Enable OR NOT DriveReady OR ErrorData.ErrorType = E_ErrorType.ERROR THEN	  
			DriveRun := FALSE;
			eTakeOverState := E_TakeOverState.STOP;
			
			IF iListener <> 0 THEN
			   iListener.M_TakeoverStopEvent();
		   	END_IF

		// Regular takeover complete if previous position completed handover
		ELSIF PrevTransportData.rTransportControlData.eHandOverState = E_HandOverState.COMPLETE THEN
			DriveRun := FALSE;
			eTakeOverState := E_TakeOverState.COMPLETE;
			
			IF iListener <> 0 THEN
			   iListener.M_TakeoveCompleteEvent();
		   	END_IF

		// End takeover and clear TU data index if abort is requested
		ELSIF AbortTakeover THEN
			DeletePrevTransportData := TRUE;
			DriveRun := FALSE;
			eTakeOverState := E_TakeOverState.COMPLETE;
		END_IF

	
(*************************************************************************
  Stop
*************************************************************************)
	E_TakeOverState.STOP:
		TakeoverOngoing := TRUE;

		// If the previous position aborted the handover or the link is broken, cancel the started takeover
		IF PrevTransportData.rTransportControlData.eHandOverState = E_HandOverState.IDLE OR
		   PrevTransportData.rTransportControlData.eHandOverState = E_HandOverState.UNDEFINED THEN

		  	IF iListener <> 0 THEN
				iListener.M_PrevUnlinkedEvent();
		   	END_IF
			
			DeletePrevTransportData := TRUE;
			eTakeOverState := E_TakeOverState.IDLE;
			
			// Send debug message
			DebugMsg := 'STOP - Takeover canceled';
			fbDebugMsg.M_SendInfoMsg(DebugMsg);				  
					
		// If the position is enabled
		ELSIF Enable THEN
			// No error is pending
			IF ErrorData.ErrorType <> E_ErrorType.ERROR THEN
				IF DriveReady THEN
					DriveRun := TRUE;
					DriveRequest := FALSE;
					eTakeOverState := E_TakeOverState.ACTIVE;
				ELSE
					DriveRequest := TRUE;
				END_IF
			END_IF
		END_IF


(*************************************************************************
  Interrupted
*************************************************************************)
	E_TakeOverState.INTERRUPTED:
		TakeoverOngoing := TRUE;
		// If the stop from the previous position is no longer required
		IF PrevTransportData.rTransportControlData.eHandOverState <> E_HandOverState.STOP THEN
			eTakeOverState := E_TakeOverState.ACTIVE;
		END_IF


(*************************************************************************
  Complete
*************************************************************************)
	E_TakeOverState.COMPLETE:
		TakeoverOngoing := FALSE;
		DriveRun := FALSE;
		// Transfer complete at prvious zone
		IF PrevTransportData.rTransportControlData.eHandOverState <> E_HandOverState.COMPLETE THEN
			DeletePrevTransportData := TRUE;
			eTakeOverState := E_TakeOverState.IDLE;
		END_IF


(*************************************************************************
  State error
*************************************************************************)
ELSE
	// Set error
	F_SetError(	
		ErrorType	:= E_ErrorType.ERROR,
		ErrorParam	:= INT_TO_STRING(eTakeOverState),
		ErrorMsg	:= E_ErrorConv.SOFTWARE_ERROR,
		ErrorData	:= ErrorData);
END_CASE

ePrevHandOverState := PrevTransportData.rTransportControlData.eHandOverState;

/// Initialize module
METHOD M_Init : BOOL // Returns true if successful, otherwise false
VAR_INPUT
END_VAR
eTakeOverState := E_TakeOverState.IDLE;
DeletePrevTransportData := FALSE;
RequestPrevTransportData := FALSE;

M_Init := TRUE;
END_METHOD

END_FUNCTION_BLOCK

// ---- 20_Product/10_BCF/11_Conv/12_E_Functions/10_Helper/F_MoveTU_DataIndex.TcPOU
FUNCTION F_MoveTU_DataIndex : DINT
(**************************************************************************************
 * 	Application		:	BoxControl Framework
 *	Revision		:	$Revision: 404529 $
 *	Revision date	:	$Date: 2018-04-23 08:21:38 +0200 (Mo., 23 Apr 2018) $
 *	Last changed by	:	$Author: b7bolm $
 *	URL				:	$URL: http://almscdc.swisslog.com/repo/SWPD/Development/BoxControlFramework/20_Release/trunk/01_Software/BCF/BCF/JumpStart/20_Product/10_App/12_E_Functions/10_Lib/10_Conv/10_Functions/F_MoveTU_DataIndex.TcPOU $
 *
 *	Purpose			:	Moves TU data from a position.
 *
 * ------------------------------------------------------------------------------------
 *	Copyright Swisslog [IP AG], Switzerland. All rights reserved.
 * 
 * ------------------------------------------------------------------------------------
 *	
 * 	Revision History: 
 *
 * 	VERSION			DATE			INITIALS			DESCRIPTION
 *	0.1				01.01.2001		swl					Example
 *
 **************************************************************************************)
VAR_INPUT
	eFunctionNumber	: E_FunctionNumber; // Function number of corresponding function
	mZoneNumber 	: INT; // Zone number
END_VAR

VAR
	STI_Instance	: ITF_SubsystemTransport; // Instance to compare valid interfaces
END_VAR

// Check if function number is valid
IF eFunctionNumber > E_FunctionNumber.F_BEGIN_FUNCTION AND
   eFunctionNumber < E_FunctionNumber.F_END_FUNCTION THEN
  
	// Check reference is valid
	IF __ISVALIDREF(FunctionRegistry[eFunctionNumber].rFunction) THEN
   		// Return tu data index
   		F_MoveTU_DataIndex := FunctionRegistry[eFunctionNumber].rFunction.M_MoveTU_DataIndex(mZoneNumber := mZoneNumber);
	END_IF
	
ELSIF eFunctionNumber > E_FunctionNumber.F_BEGIN_EXTERN_FUNCTION AND
	  eFunctionNumber < E_FunctionNumber.F_END_EXTERN_FUNCTION THEN
	  
	// Check interface is valid
	IF __QUERYINTERFACE(fbSTI_Channels[eFunctionNumber].Instance,STI_Instance) THEN
		// Return tu data index
		F_MoveTU_DataIndex := fbSTI_Channels[eFunctionNumber].Instance.M_MoveTU_DataIndex();
	END_IF
END_IF

END_FUNCTION

// ---- 20_Product/10_BCF/11_Conv/12_E_Functions/10_Helper/FB_TakeoverTracking.TcPOU
FUNCTION_BLOCK FB_TakeoverTracking IMPLEMENTS I_TakeoverListener
(**************************************************************************************
* Application : BoxControl Framework 
* Revision date : $Date: 2021-04-01 10:33:04 +0200 (tor, 01 apr 2021) $
* Author : CDC
* ------------------------------------------------------------------------------------ 
* © Swisslog AG 
* Swisslog is not liable for any usage of this source code that is not agreed 
* on between Swisslog and the other party. The mandatory legal liability remains 
* unaffected. 
* ------------------------------------------------------------------------------------ 
* Project revision history: 
* 
* 	VERSION 		DATE 			INITIALS 			DESCRIPTION 
* 	0.1 			31.08.2018 		ahe 				First implementation
* 
**************************************************************************************)
VAR_INPUT
	Param 						: ST_TransportControlParam; // Parameter of the transport control
	PrevTransportData  			: ST_TransportData; // Previous transport data
	Enable						: BOOL; // Transport enable
	EnableTakeOver 				: BOOL; // Transport enable takeover 
	StartTrackingSensor			: BOOL; // Start tracking Sensor
	StartTrackingPosition		: UDINT; // Position of start tracking sensor [mm]
	DriveReady					: BOOL;  // Drive is ready to be switched on
	EncoderValueInc				: UDINT; // Encoder value [mm]
	MaxEncoderValueInc			: UDINT; // Max encoder value [mm]
	RateIncPerMM				: LREAL; // Resolution amount of inc per mm
	iWindowTracking				: I_WindowTracking;  // Window tracking implementation
END_VAR
VAR_OUTPUT
	DriveRun   				 	: BOOL; // Run signal for drive
	DriveStop   			 	: BOOL; // Stop signal for drive
	RequestPrevTransportData 	: BOOL; // Request previous transport data
	DeletePrevTransportData	 	: BOOL; // Delete previous transport data
	Initialized					: BOOL; // Module is initialized
	eTakeOverState 				: E_TakeoverState; // Current takeover state
	ePrevHandOverState			: E_HandOverState; // Previous handover state
	TakeoverOngoing				: BOOL; // A takeover is ongoing, statemachine in operation
	TakingOverTU				: BOOL; // True when TU is being handed over and has not reached start tracking sensor yet.
END_VAR
VAR_IN_OUT
	ZoneData					: ST_ZoneData; // Zone data
	ErrorData 					: ST_ErrorDataSet; // Error data
END_VAR
VAR
	fbDebugMsg					: FB_DebugMsg; // Debug instance
	DebugMsg					: T_MAXSTRING; // Debug message
	fbTimeoutTake 				: FB_DisplacementMeter; // Timeout take
	TimeoutTakeDistance			: DINT; // Distance until timeout take is triggered [mm]
	TransitionTU_DataIndex 		: DINT; // Transition TU-data index at takeover from previous zone to tracking
	TrackingZoneIndex			: UINT; // Tracking zone index
	TrackingZoneIndexRE			: UINT; // Tracking zone index rear edge
	eTrackingState				: E_TakeoverTrackingState; // Tracking state machine
	TransportEnable				: BOOL; // Hardstop 
	TransportEnableTakeOver		: BOOL; // Softstop takeover
	TU_InTransition				: BOOL; // Tu is between takeover and start tracking
	fbTakeover 					: FB_Takeover; // Takeover control
	CreateGap					: BOOL; // Command to create gap
	fbGapMeter					: FB_DisplacementMeter; // Distance meter to create minimal gap between TUs
	DrivePreStart 				: BOOL; // Drive pre start 2 zones ahead
	AbortTakeover				: BOOL; // Takeover must be aborted
END_VAR

//Input mapping
TransportEnable := Enable AND Param.rZoneEnable.Transport;
TransportEnableTakeOver := EnableTakeOver AND Param.rZoneEnable.TakeOver;

F_ResetError(Reset := FALSE, ErrorData := ErrorData);	

IF iWindowTracking = 0 THEN
	RETURN;
END_IF

// Initialization of the module
// Module initialization
IF NOT Initialized THEN
	RETURN;
END_IF

(**************************************************************************************************************
   Tracking state
***************************************************************************************************************)
CASE eTrackingState OF
	// Idle
	E_TakeoverTrackingState.WAITING_FOR_TAKEOVER:
		TakingOverTU := FALSE;
		TU_InTransition := FALSE;
		IF ZoneData.TransportControlData.eTakeOverState = E_TakeoverSTate.ACTIVE THEN
			fbTimeoutTake(Run := FALSE);
			TU_InTransition := TRUE;
			TakingOverTU := TRUE;
			
			// When an adding process at Starttracking is ongoing, wait until its finished
			IF TrackingZoneIndex > 0 THEN
				eTrackingState := E_TakeoverTrackingState.TRACKING_ALLOCATION_ONGOING;
			ELSE
				eTrackingState := E_TakeoverTrackingState.DETECT_TU_FRONTEDGE;
			END_IF
		END_IF
		
	// Adding process still ongoing, wait until start tracking is free to add new one
	E_TakeoverTrackingState.TRACKING_ALLOCATION_ONGOING:
		IF TrackingZoneIndex = 0 THEN
			eTrackingState := E_TakeoverTrackingState.DETECT_TU_FRONTEDGE;
		END_IF
		TakingOverTU := FALSE;
		
	E_TakeoverTrackingState.DETECT_TU_FRONTEDGE:
		// Run timeout start tracking
		fbTimeoutTake(
			Run 				:= TRUE, 
			EncoderValueInc		:= EncoderValueInc,
			MaxEncoderValueInc 	:= MaxEncoderValueInc,
			RateIncPerMM		:= RateIncPerMM,
			SetPoint 			:= TimeoutTakeDistance);
	
		// Wait until TU arrives at start tracking sensor
		IF StartTrackingSensor THEN
			TrackingZoneIndex := iWindowTracking.M_AddTU_FE(
									mTU_Index			:= TransitionTU_DataIndex, 
									mAbsolutePosition	:= StartTrackingPosition, 
									miActionListener	:= 0);
		
			IF TrackingZoneIndex > 0 THEN
				eTrackingState := E_TakeoverTrackingState.FINISH_TAKEOVER;
			ELSE
				DebugMsg := 'Fatal error - New TU FE could not be added to WindowTracking';
				fbDebugMsg.M_SendInfoMsg(DebugMsg);	
				eTrackingState := E_TakeoverTrackingState.WAITING_FOR_TAKEOVER;
			END_IF
			
			TU_InTransition := FALSE;
			TakingOverTU := FALSE;

		ELSIF fbTimeoutTake.Q THEN
			fbTimeoutTake(Run := FALSE);
			
			// Send debug message
			DebugMsg := CONCAT('Timeout start tracking, TU did not show up at start tracking sensor', Param.rSettings.ZoneName);
			fbDebugMsg.M_SendInfoMsg(DebugMsg);	
			
			TU_InTransition := FALSE;
			TakingOverTU := FALSE;
			AbortTakeover := TRUE;
			M_DeleteTU_DataIndex();
			
			eTrackingState := E_TakeoverTrackingState.FINISH_TAKEOVER;
		END_IF
		
	// WAITING_TRANSPORT_FINISHED
	E_TakeoverTrackingState.FINISH_TAKEOVER:
		fbTimeoutTake();
		
		IF ZoneData.TransportControlData.eTakeOverState <> E_TakeoverSTate.ACTIVE AND 
           ZoneData.TransportControlData.eTakeOverState <> E_TakeoverSTate.COMPLETE THEN
			AbortTakeover := FALSE;
			eTrackingState := E_TakeoverTrackingState.WAITING_FOR_TAKEOVER;
			
		ELSIF fbTimeoutTake.Q THEN
			fbTimeoutTake(Run := FALSE);
			
			// Send debug message
			DebugMsg := CONCAT('Timeout takeover, handshake not completed', Param.rSettings.ZoneName);
			fbDebugMsg.M_SendInfoMsg(DebugMsg);	
			
			AbortTakeover := TRUE;
			M_DeleteTU_DataIndex();
		END_IF
ELSE
	eTrackingState := E_TakeoverTrackingState.WAITING_FOR_TAKEOVER;
END_CASE

(**************************************************************************************************************
   Complete adding process 
   When a TU was detected at start tracking, wait for rear edge to complete
***************************************************************************************************************)
IF TrackingZoneIndex > 0 THEN
	IF NOT StartTrackingSensor THEN
		TrackingZoneIndexRE := iWindowTracking.M_AddTU_RE(
									mAbsolutePosition	:= StartTrackingPosition, 
									mZoneIndex			:= TrackingZoneIndex);
									
		// When the adding was completet successfully
		IF TrackingZoneIndexRE > 0 THEN
			;
		ELSE
			DebugMsg := 'Fatal error - New TU RE could not be added to WindowTracking';
			fbDebugMsg.M_SendInfoMsg(DebugMsg);	
		END_IF
		
		TrackingZoneIndex := 0;
	END_IF
END_IF

(**************************************************************************************************************
   Create minimum gap between TUs
***************************************************************************************************************)
IF eTakeOverState = E_TakeOverState.ACTIVE THEN
	CreateGap := TRUE;
END_IF

IF Param.rSettings.MinimumTU_Distance > 0 THEN 
	IF CreateGap AND eTakeOverState = E_TakeOverState.IDLE THEN
		fbGapMeter(
			Run					:= TRUE, 
			EncoderValueInc		:= EncoderValueInc,
			MaxEncoderValueInc 	:= MaxEncoderValueInc,
			RateIncPerMM 		:= RateIncPerMM,
			SetPoint			:= Param.rSettings.MinimumTU_Distance);
	END_IF
ELSE
	CreateGap := FALSE;
END_IF

fbGapMeter( 
	EncoderValueInc		:= EncoderValueInc,
	MaxEncoderValueInc 	:= MaxEncoderValueInc,
	RateIncPerMM 		:= RateIncPerMM);
	
IF fbGapMeter.Q THEN
	fbGapMeter(Run := FALSE);
	CreateGap := FALSE;
END_IF

(**************************************************************************************************************
   Takeover state
***************************************************************************************************************)
fbTakeover(
	Enable					:= TransportEnable AND
            		   		  (Param.rOperationState.eState = E_PositionState.STARTED OR
	         		    	   Param.rOperationState.eState = E_PositionState.STOPPING),
	RequestTakeover			:= Param.rOperationState.eState = E_PositionState.STARTED AND
							   TransportEnableTakeOver AND
							   NOT TU_InTransition AND
							   NOT CreateGap,						   
	AbortTakeover 			:= AbortTakeover,
	PrevZonePresent			:= Param.rePrevFunctionNumber > 0,
	EncoderValue			:= EncoderValueInc,
	MaxEncoderValue			:= MaxEncoderValueInc,
	EncoderRate 			:= RateIncPerMM,
	DriveReady				:= DriveReady,
	iListener				:= THIS^,
	DriveRun				=> ,
	eTakeOverState			=> eTakeOverState,
	ePrevHandOverState		=> ePrevHandOverState,
	RequestPrevTransportData=> RequestPrevTransportData,
	DeletePrevTransportData	=> DeletePrevTransportData,
	TakeoverOngoing			=> TakeoverOngoing,
	PrevTransportData		:= PrevTransportData,
	ErrorData				:= ErrorData);

DrivePreStart := PrevTransportData.rTransportControlData.TransportActive AND eTakeOverState = E_TakeoverState.READY OR fbTakeover.DriveRequest;
	
DriveRun := fbTakeover.DriveRun OR CreateGap OR eTrackingState = E_TakeoverTrackingState.DETECT_TU_FRONTEDGE OR DrivePreStart;

ZoneData.TransportControlData.eTakeOverState := eTakeOverState;

DriveStop := fbTakeover.TakeoverOngoing AND NOT fbTakeover.DriveRun AND NOT fbTakeover.DriveRequest;

METHOD PROTECTED  M_DeleteTU_DataIndex

VAR_INPUT
END_VAR

VAR
  WindowTrackingIndex   : UDINT                  := 0;
END_VAR
{warning disable C0371}
IF NOT __ISVALIDREF(ZoneData) THEN
	RETURN;
END_IF

// If a TU-data index is existing 
IF TransitionTU_DataIndex <> 0 THEN
	// If TU- and assignment ID is unknown
	IF     TU_DataTable[TransitionTU_DataIndex].TU_ID.ASCII  = Conveyor.TU_ID_UNKNOWN
       AND TU_DataTable[TransitionTU_DataIndex].AssignmentID = Conveyor.ASSIGNMENT_ID_UNKNOWN THEN
		// debug message: '11-001-0095-01-1,  unknown TU_DataIndex deleted,  TU_DataIndex = 5,  TuID = 000012345,  AssignmentID = 999999999'
		DebugMsg := '';
		DebugMsg := CONCAT(DebugMsg, F_AddDividerToSisString(Param.rSettings.ZoneName));
		DebugMsg := CONCAT(DebugMsg, ',  unknown TU_DataIndex deleted');
		DebugMsg := CONCAT(DebugMsg, F_CreateTU_DataString(TU_DataIndex:= TransitionTU_DataIndex));
		// Delete TU-data
		F_DeleteTU_Data(
			TU_DataIndex	:= TransitionTU_DataIndex,
			NoTTC 			:= FALSE);

		// delete TU index from window tracking
		WindowTrackingIndex:= iWindowTracking.M_GetZoneIndex(mAbsolutePosition:= StartTrackingPosition);
		IF WindowTrackingIndex > 0 THEN
			IF iWindowTracking.P_ZoneTable[WindowTrackingIndex].TU_Index = TransitionTU_DataIndex THEN
				iWindowTracking.P_ZoneTable[WindowTrackingIndex].TU_Index:= 0;
			END_IF
		END_IF
	END_IF

	// Update last TU data index			
	IF TransitionTU_DataIndex <> 0 THEN
		ZoneData.TransportControlData.LastTU_DataIndex := ZoneData.TransportControlData.TU_DataIndex;
	END_IF		

	// Update states
	TransitionTU_DataIndex := 0;
	ZoneData.TransportControlData.DataPresent := FALSE;
END_IF
{warning restore C0371}
END_METHOD

/// Initialize Takeover tracking
METHOD M_Init : BOOL
fbTakeover.M_Init();
eTrackingState := E_TakeoverTrackingState.WAITING_FOR_TAKEOVER;

fbTimeoutTake(Run := FALSE);

// Timeout take monitoring
IF Param.rSettings.TimeoutTakeDistance <> 0 THEN
	TimeoutTakeDistance := Param.rSettings.TimeoutTakeDistance;
ELSE
	TimeoutTakeDistance := 3000;
END_IF

CreateGap := TRUE;

Initialized := TRUE;

M_Init := TRUE;
END_METHOD

METHOD M_PrevUnlinkedEvent
M_DeleteTU_DataIndex();
END_METHOD

METHOD M_TakeoveCompleteEvent
END_METHOD

METHOD M_TakeoverStartEvent
END_METHOD

METHOD M_TakeoverStopEvent
VAR_INPUT
END_VAR
END_METHOD

METHOD M_TU_IndexMovedEvent
VAR_INPUT
	mMovedTU_Index	: DINT;
END_VAR

IF mMovedTU_Index > 0 THEN
	// Delete TU-data if it is configured
	IF Param.rSettings.DeleteTU_DataTakeover THEN
		// debug message: '11-001-0095-01-1,  moved TU_DataIndex deleted,  TU_DataIndex = 5,  TuID = 000012345,  AssignmentID = 999999999'
		DebugMsg := '';
		DebugMsg := CONCAT(DebugMsg, F_AddDividerToSisString(Param.rSettings.ZoneName));
		DebugMsg := CONCAT(DebugMsg, ',  moved TU_DataIndex deleted');
		DebugMsg := CONCAT(DebugMsg, F_CreateTU_DataString(TU_DataIndex:= mMovedTU_Index));
		fbDebugMsg.M_SendInfoMsg(DebugMsg);
		// If data has been deleted
		If F_DeleteTU_Data(
			TU_DataIndex 	:= mMovedTU_Index,
			NoTTC 			:= FALSE) THEN
	
			M_DeleteTU_dataIndex();
		END_IF
	END_IF
END_IF

TransitionTU_DataIndex := mMovedTU_Index;
END_METHOD

END_FUNCTION_BLOCK

// ---- 20_Product/10_BCF/11_Conv/12_E_Functions/10_Helper/FB_TakeoverTrackingMerge.TcPOU
/// Functionality to control a takeover process onto a tracking conveyor
FUNCTION_BLOCK FB_TakeoverTrackingMerge IMPLEMENTS I_TakeoverListener
(************************************************************************************** 
* 	Application 		: BoxControl Framework 
* 	Revision 			: $Revision: 408723 $ 
* 	Revision date 		: $Date: 2018-06-27 13:49:08 +0200 (Wed, 27 Jun 2018) $ 
* 	Last changed by 	: $Author: b7bolm $ 
* 	URL 				: $URL: http://almscdc.swisslog.com/repo/SWPD/Development/BoxControlFramework/21_Projects/BCF_2.0/trunk/BCF/BCF/JumpStart/20_Product/10_App/12_E_Functions/10_Lib/10_Conv/FB_FunctionList.TcPOU $ 
* ------------------------------------------------------------------------------------ 
* 	© Swisslog AG 
* 	Swisslog is not liable for any usage of this source code that is not agreed 
* 	on between Swisslog and the other party. The mandatory legal liability remains 
* 	unaffected. 
* ------------------------------------------------------------------------------------ 
* 	Revision History: 
* 
* 	VERSION 		DATE 			INITIALS 			DESCRIPTION 
* 	0.1 			31.08.2018 		ahe 				First implementation
*	0.2				12.11.2018		mbo					Review
*	0.3				01.04.2021		ahe					Added timeout takeover
* 
**************************************************************************************)
VAR_INPUT
	Param 							: ST_TransportControlParam; // Parameter of the transport control
	PrevTransportData  				: ST_TransportData; // Previous transport data
	Enable							: BOOL; // Transport enable
	EnableTakeOver 					: BOOL; // Transport enable takeover 
	ActionId						: INT; // ID of this action for tracking purposes
	TU_Length						: UINT; // TU length to be allocated on tracking
	FrontGap						: UINT; // Gap between zone start and TU
	RearGap							: UINT; // Gap between zone end and TU
	MergingPosition					: UDINT; // Merging position on tracking
	MergingTolerance				: UDINT; // Merging tolerance to allow merging
	DriveCompleteDelayDistance		: DINT;  // Delay drive distance when takeover is complete
	DriveStopDelayDistance			: DINT;  // Delay drive distance when takeover is stopped
	DriveReady						: BOOL;  // Drive is ready to be switched on
	EncoderValueInc					: UDINT; // Encoder value [inc]
	MaxEncoderValueInc				: UDINT; // Max encoder value [inc]
	RateIncPerMM					: LREAL; // Resolution amount of incs per mm
	iWindowTracking					: I_WindowTracking;  // Window tracking implementation
END_VAR
VAR_OUTPUT
	DriveRun   				 		: BOOL; // Run signal for drive
	DriveStop   			 		: BOOL; // Stop signal for drive
	RequestPrevTransportData 		: BOOL; // Request previous transport data
	DeletePrevTransportData	 		: BOOL; // Delete previous transport data
	Initialized						: BOOL; // Module is initialized
	eTakeOverState 					: E_TakeoverState; // Current takeover state
	ePrevHandOverState				: E_HandOverState; // Previous handover state
	AvailableZoneIndex				: UINT; // Current available valid Zone index
	TakeoverOngoing					: BOOL; // A takeover is ongoing, statemachine in operation
END_VAR
VAR_IN_OUT
	ZoneData						: ST_ZoneData; // Zone data
	ErrorData 						: ST_ErrorDataSet; // Error data
END_VAR
VAR
	fbDebugMsg						: FB_DebugMsg; // Debug instance
	DebugMsg						: T_MAXSTRING; // Debug message
	fbTimeoutTake 					: FB_DisplacementMeter; // Timeout take
	TimeoutTakeDistance				: DINT; // Distance until timeout take is triggered [mm]
	TransportEnable					: BOOL; // Hardstop 
	TransportEnableTakeOver			: BOOL; // Softstop takeover
	fbTakeover 						: FB_Takeover; // Takeover control
	TrackingZoneIndex				: UINT; // Tracking zone index
	DistanceToZone					: DINT; // Distance to zone from merging point
	DriveDelayActive				: BOOL; // Drive delay is currently active
	LastZoneIndex 					: UINT; // Last zone where  a TU was added
	LastTU_Index 					: DINT; // Last TU index which was added to a zone
	fbDriveDelayMeter				: FB_DisplacementMeter; // Distance meter to create minimal gap between TUs
	AbortTakeover					: BOOL; // Takeover must be aborted
END_VAR

//Input mapping
TransportEnable := Enable AND Param.rZoneEnable.Transport;
TransportEnableTakeOver := EnableTakeOver AND Param.rZoneEnable.TakeOver;

F_ResetError(Reset := FALSE, ErrorData := ErrorData);	

IF iWindowTracking = 0 OR 
   ActionId = 0 OR 
   TU_Length = 0 THEN
	RETURN;
END_IF

// Initialization of the module
// Module initialization
IF NOT Initialized THEN
	RETURN;
END_IF

(**************************************************************************************************************
   Determine zone for this position
***************************************************************************************************************)
AvailableZoneIndex := 0;

// Wait until a zone can be found at merging point
TrackingZoneIndex := iWindowTracking.M_GetZoneIndex(MergingPosition);
	
// When a possible zone was found, validate and monitor it.
IF TrackingZoneIndex > 0 THEN
	// As long the zone is valid
	IF iWindowTracking.P_ZoneTable[TrackingZoneIndex].Used THEN
		// Zone gets monitored as long it is in a certain range 
		DistanceToZone := iWindowTracking.M_GetDistanceToZoneStart(MergingPosition, TrackingZoneIndex);

		IF ABS(DistanceToZone + FrontGap) <= UDINT_TO_DINT(MergingTolerance) THEN
			// When zone is assigned to this position and is empty,
			// Zone is a possible next to be merged
			IF NOT iWindowTracking.P_ZoneTable[TrackingZoneIndex].TU_Present AND
			   iWindowTracking.P_ZoneTable[TrackingZoneIndex].ActionId = ActionId THEN
				// As a reason that a position can reserve zones for different TU lengths
				// length of zone should be compared.
				IF iWindowTracking.P_ZoneTable[TrackingZoneIndex].ZoneLength >= TU_Length + FrontGap + RearGap THEN
					AvailableZoneIndex := TrackingZoneIndex;
				END_IF
			END_IF
		ELSE
			TrackingZoneIndex := 0;
		END_IF
	ELSE
		TrackingZoneIndex := 0;
	END_IF
END_IF

(**************************************************************************************************************
   Delay drive to complete handover to tracked conveyor
   Active when takeover was successfully completed.
***************************************************************************************************************)
fbDriveDelayMeter( 
	EncoderValueInc		:= EncoderValueInc,
	MaxEncoderValueInc 	:= MaxEncoderValueInc,
	RateIncPerMM		:= RateIncPerMM);

IF fbDriveDelayMeter.Q THEN
	DriveDelayActive := FALSE;
	fbDriveDelayMeter(Run := FALSE);
END_IF
	
(**************************************************************************************************************
   Takeover state
***************************************************************************************************************)
fbTimeoutTake(
	EncoderValueInc		:= EncoderValueInc,
	MaxEncoderValueInc 	:= MaxEncoderValueInc,
	RateIncPerMM		:= RateIncPerMM);
	
// Timeout take happened
IF fbTimeoutTake.Q THEN
	fbTimeoutTake(Run := FALSE);
	M_TimeoutTakeEvent();
	AbortTakeover := TRUE;
	
	// Send debug message
	DebugMsg := CONCAT('Timeout takeover, takeover was not completed', Param.rSettings.ZoneName);
	fbDebugMsg.M_SendInfoMsg(DebugMsg);
END_IF
						
fbTakeover(
	Enable					:= TransportEnable AND 
            				  (Param.rOperationState.eState = E_PositionState.STARTED OR
	         				   Param.rOperationState.eState = E_PositionState.STOPPING), 
	RequestTakeover			:= Param.rOperationState.eState = E_PositionState.STARTED AND
							   TransportEnableTakeOver AND 
							   AvailableZoneIndex <> 0,
	AbortTakeover 			:= AbortTakeover,
	PrevZonePresent			:= Param.rePrevFunctionNumber > 0,
	EncoderValue			:= EncoderValueInc, 
	MaxEncoderValue			:= MaxEncoderValueInc,
	EncoderRate 			:= RateIncPerMM,
	DriveReady				:= DriveReady,
	iListener				:= THIS^,
	eTakeOverState			=> eTakeOverState, 
	ePrevHandOverState		=> ePrevHandOverState, 
	RequestPrevTransportData=> RequestPrevTransportData,
	DeletePrevTransportData	=> DeletePrevTransportData,
	TakeoverOngoing			=> TakeoverOngoing,
	PrevTransportData		:= PrevTransportData,
	ErrorData				:= ErrorData);
	
DriveRun := fbTakeover.DriveRun OR (DriveDelayActive AND DriveReady);

ZoneData.TransportControlData.eTakeOverState := eTakeOverState;

DriveStop := fbTakeover.TakeoverOngoing AND NOT fbTakeover.DriveRun AND NOT fbTakeover.DriveRequest;

METHOD PROTECTED  M_DeleteTU_DataIndex : BOOL
VAR_INPUT
	mTU_Index	: DINT;
END_VAR
M_DeleteTU_DataIndex := FALSE;
// If a TU-data index is existing 
IF mTU_Index <> 0 THEN
	// If TU-ID is unknown
	IF TU_DataTable[mTU_Index].TU_ID.ASCII = Conveyor.TU_ID_UNKNOWN THEN
		// debug message: '11-001-0095-01-1,  unknown TU_DataIndex deleted,  TU_DataIndex = 5,  TuID = 000012345,  AssignmentID = 999999999'
		DebugMsg := '';
		DebugMsg := CONCAT(DebugMsg, F_AddDividerToSisString(Param.rSettings.ZoneName));
		DebugMsg := CONCAT(DebugMsg, ',  unknown TU_DataIndex deleted');
		DebugMsg := CONCAT(DebugMsg, F_CreateTU_DataString(TU_DataIndex:= mTU_Index));
		fbDebugMsg.M_SendErrorMsg(DebugMsg);
		// Delete TU-data
		M_DeleteTU_DataIndex := F_DeleteTU_Data(
									TU_DataIndex	:= mTU_Index,
									NoTTC 			:= FALSE);
	END_IF
END_IF
END_METHOD

/// Initialize Takeover tracking
METHOD M_Init : BOOL
fbTakeover.M_Init();

fbTimeoutTake(Run := FALSE);

// Timeout take monitoring
IF Param.rSettings.TimeoutTakeDistance <> 0 THEN
	TimeoutTakeDistance := Param.rSettings.TimeoutTakeDistance;
ELSE
	TimeoutTakeDistance := 3000;
END_IF

Initialized := TRUE;

M_Init := TRUE;
END_METHOD

METHOD M_PrevUnlinkedEvent
VAR
	mTU_Index 		: DINT;
END_VAR
mTU_Index := 0;

// When window tracking is avialable and a last known index
IF iWindowTracking <> 0 THEN
	IF LastZoneIndex > 0 THEN
		// Ensure zone is sitll part of this zone
		IF iWindowTracking.P_ZoneTable[LastZoneIndex].Used AND
		   iWindowTracking.P_ZoneTable[LastZoneIndex].TU_Present AND
		   iWindowTracking.P_ZoneTable[LastZoneIndex].ActionId = ActionId AND
           iWindowTracking.P_ZoneTable[LastZoneIndex].TU_Index = LastTU_Index THEN
		   
		   // Clear only TU index and keep zone allocation.
		   // Remark: It is not 100% clear what was happening with the physical TU
		   // Therefore the zone allocation is kept but the link the TU Data is cleared
		   // to prevent data inconsistency.
		   mTU_Index := iWindowTracking.P_ZoneTable[LastZoneIndex].TU_Index;
		   
		   iWindowTracking.P_ZoneTable[LastZoneIndex].TU_Index := 0;
		END_IF
	END_IF
END_IF

IF mTU_Index > 0 THEN
	M_DeleteTU_DataIndex(mTU_Index);
END_IF
END_METHOD

METHOD M_TakeoveCompleteEvent
fbTimeoutTake(Run := FALSE);
fbDriveDelayMeter(Run := FALSE);
fbDriveDelayMeter(
	Run					:= TRUE, 
	EncoderValueInc		:= EncoderValueInc,
	MaxEncoderValueInc 	:= MaxEncoderValueInc,
	RateIncPerMM		:= RateIncPerMM,
	SetPoint			:= DriveCompleteDelayDistance);
	
DriveDelayActive := TRUE;
END_METHOD

METHOD M_TakeoverStartEvent
AbortTakeover := FALSE;
fbTimeoutTake(Run := FALSE);

// Run timeout start tracking
fbTimeoutTake(
	Run 				:= TRUE,
	SetPoint 			:= TimeoutTakeDistance);
END_METHOD

METHOD M_TakeoverStopEvent
VAR_INPUT
END_VAR
IF DriveStopDelayDistance > 0 THEN
	fbDriveDelayMeter(Run := FALSE);
	fbDriveDelayMeter(
		Run					:= TRUE, 
		EncoderValueInc		:= EncoderValueInc,
		MaxEncoderValueInc 	:= MaxEncoderValueInc,
		RateIncPerMM		:= RateIncPerMM,
		SetPoint			:= DriveStopDelayDistance);
		
	DriveDelayActive := TRUE;
ELSE
	DriveDelayActive := FALSE;
END_IF
END_METHOD

METHOD M_TimeoutTakeEvent
VAR
	mTU_Index 		: DINT;
END_VAR
mTU_Index := 0;

// When window tracking is avialable and a last known index
IF iWindowTracking <> 0 THEN
	IF LastZoneIndex > 0 THEN
		// Ensure zone is sitll part of this zone
		IF iWindowTracking.P_ZoneTable[LastZoneIndex].Used AND
		   iWindowTracking.P_ZoneTable[LastZoneIndex].TU_Present AND
		   iWindowTracking.P_ZoneTable[LastZoneIndex].ActionId = ActionId AND
           iWindowTracking.P_ZoneTable[LastZoneIndex].TU_Index = LastTU_Index THEN
		   
		   // Clear only TU index and keep zone allocation.
		   // Remark: It is not 100% clear what was happening with the physical TU
		   // Therefore the zone allocation is kept but the link the TU Data is cleared
		   // to prevent data inconsistency.
		   mTU_Index := iWindowTracking.P_ZoneTable[LastZoneIndex].TU_Index;
		   
		   iWindowTracking.P_ZoneTable[LastZoneIndex].TU_Index := 0;
		END_IF
	END_IF
END_IF

IF mTU_Index > 0 THEN
	M_DeleteTU_DataIndex(mTU_Index);
END_IF
END_METHOD

METHOD M_TU_IndexMovedEvent
VAR_INPUT
	mMovedTU_Index	: DINT;
END_VAR
VAR_INST
	AddTU_Ok		: BOOL;
END_VAR
IF mMovedTU_Index > 0 THEN
	// Delete TU-data if it is configured
	IF Param.rSettings.DeleteTU_DataTakeover THEN
		// debug message: '11-001-0095-01-1,  moved TU_DataIndex deleted,  TU_DataIndex = 5,  TuID = 000012345,  AssignmentID = 999999999'
		DebugMsg := '';
		DebugMsg := CONCAT(DebugMsg, F_AddDividerToSisString(Param.rSettings.ZoneName));
		DebugMsg := CONCAT(DebugMsg, ',  moved TU_DataIndex deleted');
		DebugMsg := CONCAT(DebugMsg, F_CreateTU_DataString(TU_DataIndex:= mMovedTU_Index));
		fbDebugMsg.M_SendErrorMsg(DebugMsg);
		// If data has been deleted
		IF F_DeleteTU_Data(
				TU_DataIndex 	:= mMovedTU_Index,
				NoTTC 			:= FALSE) THEN
			
			M_DeleteTU_DataIndex(mMovedTU_Index);			
			mMovedTU_Index := 0;
		END_IF
	END_IF
END_IF

// When a window tracking instance is available
IF iWindowTracking <> 0 THEN
	// When a possible zone is availble, add TU to that zone
	IF AvailableZoneIndex > 0 THEN
		AddTU_Ok := iWindowTracking.M_AddTU(
						mZoneIndex 	:= AvailableZoneIndex,
						mTU_Index 	:= mMovedTU_Index,
						mLength 	:= TU_Length,
						mTU_Offset 	:= FrontGap);
		
		// Store last zone index for error handling
		LastZoneIndex := AvailableZoneIndex;
		LastTU_Index := mMovedTU_Index;
		
		IF NOT AddTU_Ok THEN
			DebugMsg := CONCAT('M_TU_IndexMovedEvent - Could not add TU to ZoneIndex:', UINT_TO_STRING(AvailableZoneIndex));
			DebugMsg := CONCAT(', Length of Zone:', UINT_TO_STRING(iWindowTracking.P_ZoneTable[AvailableZoneIndex].ZoneLength));
			DebugMsg := CONCAT(', Length of TU:', UINT_TO_STRING(TU_Length));
			fbDebugMsg.M_SendErrorMsg(DebugMsg);
		END_IF
	END_IF
END_IF
END_METHOD

END_FUNCTION_BLOCK

// ---- 20_Product/10_BCF/11_Conv/12_E_Functions/10_Helper/FB_TransportControl.TcPOU
 FUNCTION_BLOCK FB_TransportControl
(**************************************************************************************
 * 	Application		:	BoxControl Framework
 *	Revision		:	$Revision: 475083 $
 *	Revision date	:	$Date: 2021-04-10 12:07:10 +0200 (lör, 10 apr 2021) $
 *	Last changed by	:	$Author: d7mangc $
 *	URL				:	$URL: http://almscdc.swisslog.com/repo/SWPD/Development/BoxControlFramework/20_Release/tags/R1.12.0/01_Software/BCF/BCF/JumpStart/20_Product/10_BCF/11_Conv/12_E_Functions/10_Helper/FB_TransportControl.TcPOU $
 *
 *	Purpose			:	The transport control is responsible for the coordinated
 *                      physical TU and logical data movement and ensures the relation
 *                      to the position.
 *
 * ------------------------------------------------------------------------------------
 *	Copyright Swisslog [IP AG], Switzerland. All rights reserved.
 * 
 * ------------------------------------------------------------------------------------
 *	
 * 	Revision History: 
 *
 *  VERSION DATE         INITIALS     DESCRIPTION
 *  0.0     DD.MM.YYYY   (name)       (explain customized modifications)
 *
 **************************************************************************************)
VAR_INPUT
	Param 						: ST_TransportControlParam; // Parameter of the transport control
	PrevTransportData  			: ST_TransportData; // Previous transport data
	NextTransportData			: ST_TransportData; // Next transport data
	TransportEnable				: BOOL; // Transport enable
	TransportEnableTakeOver 	: BOOL; // Transport enable takeover 
	TransportEnableHandOver 	: BOOL; // Transport enable handover
	EnableFastSpeed 			: BOOL; // Enable fast speed
	ZoneOccupied 				: BOOL; // Input zone occupied
	DriveRunning				: BOOL; // Feedback drive is running
	DriveReady					: BOOL := TRUE; // Drive is ready to be started
	CurrentSpeed				: INT; // Current speed [mm/s]
	Acceleration    			: INT; // Acceleration [mm/s^2]
	StoppingDistance			: UINT; // Distance until the TU is stopped [mm]
	EncoderValue				: UDINT; // Encoder value [mm]
	MaxEncoderValue				: UDINT; // Max encoder value [mm]
	SyncTracking				: BOOL; // Trigger to sync tracking leading edge of TU to SyncTrackingPosition
	SyncTrackingPosition		: DINT; // Sync tracking leading edge position [mm]
END_VAR

VAR_OUTPUT
	Outputs						: ST_TransportControl_Outputs; // Module Internal outputs
END_VAR

VAR_IN_OUT
	ZoneData					: ST_ZoneData; // Zone data
	ErrorData 					: ST_ErrorDataSet; // Error data
END_VAR

VAR
	fbDebugMsg					: FB_DebugMsg; // Debug instance
	DebugMsg					: T_MAXSTRING; // Debug message
	Inputs 						: ST_TransportControl_Inputs; // Module internal inputs
	Init						: BOOL; // Initialized
	ZoneOccupiedSignal 			: BOOL; // Internal zone occupied signal 
	DriveFeedInRun        		: BOOL; // Switch drive on for feed in
	DriveTakeoverRun        	: BOOL; // Switch drive on for takeover
	DriveHandoverRun        	: BOOL; // Switch drive on for handover
	DriveFreeRun            	: BOOL; // Switch drive on for free run
	DriveClearingRun	    	: BOOL; // Switch drive on for clearing
	DriveMultiTU_Run	    	: BOOL; // Switch drive on for multiple TU 
	Transition_TU_DataIndex 	: DINT; // Transition TU-data index at takeover from previous zone to tracking 
    tZoneFree       			: TIME := T#2S ; // Delay time for zone occupied
	tZoneOccupied      			: TIME := T#2S; // Delay time for zone occupied	
	tAutoResetJam        		: TIME := T#2S; // Time delay auto reset jam error
   	tFreeRun             		: TIME := T#3S; // Time drive free run
    fbZoneOccupiedFreeTimer 	: FB_Timer; // Delay timer zone occupied free
    fbZoneOccupiedTimer	    	: FB_Timer; // Delay timer zone occupied
    fbFreeRunTimer          	: FB_Timer; // Timer drive free run
	fbAutoResetJamTimer     	: FB_Timer; // Timer auto reset jam error
	fbMergingServiceRetry		: FB_Timer; // Timer to retry the merging service
	fbRoutingServiceRetry		: FB_Timer; // Timer to retry the merging service
	fbTimeoutJam 				: FB_DisplacementMeter; // Timeout jam
	fbTimeoutTake 				: FB_DisplacementMeter; // Timeout take	
	fbDelayZoneOccupied			: FB_DisplacementMeter; // Delay zone occupied
	fbDelayZoneFree		 		: FB_DisplacementMeter; // Delay zone free
	fbClearing		 			: FB_DisplacementMeter; // Clearing
	fbDelayStartTakeover  		: FB_DisplacementMeter; // Delay start takeover
	fbZoneEndLengthClear		: FB_DisplacementMeter; // ZoneEndLenght clear
	fbTakeoverPlausible         : FB_DisplacementMeter; // Takever distance plausible
	DelayDistance				: DINT; // Delay distance [mm]
	TimeoutTakeDistance			: DINT; // Distance until timeout take is triggered [mm]
	StoppingByAccelaretion  	: INT; // Stopping distance by acceleration
	TU_WithinBrakingZone    	: BOOL; // The TU is within braking zone
	fbTrackingLeadingEdge 		: FB_DisplacementMeter; // TU leading edge position	tracking	
	SubsystemReg				: ST_SubsystemRegistryConv;
	TransportParam				: ST_TransportParam; // Transport parameter valid for current transport
	PrevTransportParam			: ST_TransportParam; // Previous transport parameter valid for current transport
	NextFunctionNumber			: E_FunctionNumber; // Currently assigned next function number
	EnableShortZoneRestart  	: BOOL; // Enable short zone restart
	TransportTrspDataReq    	: ST_TransportDataRequest; // TransportState, transport data request
	TakeOverTrspDataReq     	: ST_TransportDataRequest; // TakeOverState, transport data reques
	HandOverTrspDataReq     	: ST_TransportDataRequest; // HandOverState, transport data reques
	InitTrspDataReq         	: ST_TransportDataRequest; // Initial, clear structur
	SyncTrackingLeadingEdge 	: R_TRIG; // Trigger for sync tracking leading edge
	ExtSyncTrackingLeadingEdge 	: R_TRIG; // External trigger for sync tracking leading edge
	fbCascadeDrive				: TON; // Cascade drive switch on
    fbDelayTakeoverRun          : TON; // Delay timer for drive run signal requested by drive takeover run
END_VAR

VAR_STAT CONSTANT
	TIMEOUT_TAKE_FACTOR  	    : INT := 2; // Factor for timeout take setpoint
	DIST_TO_OCCUPIED			: INT := 200; // Distance before signal occupied (takeover plausibility check) [mm]
	RECALL_SERVICE_TIMEOUT      : TIME := T#2S; // Recall routing or merging service
END_VAR

(**************************************************************************************************************
   Input mapping
***************************************************************************************************************)
A_InputMapping();

(**************************************************************************************************************
   Error reset
***************************************************************************************************************)
F_ResetError(Reset := FALSE, ErrorData := ErrorData);

(**************************************************************************************************************
   Initialization
***************************************************************************************************************)
A_Init();

// Abort execution of transport control if it is not initialized
IF NOT Init THEN
	RETURN;
END_IF

(**************************************************************************************************************
   Error reset
***************************************************************************************************************)
F_ResetError(Reset := FALSE, ErrorData := ErrorData);

(**************************************************************************************************************
   Position tracking
***************************************************************************************************************)
A_PositionTracking();

(**************************************************************************************************************
   Transport state
***************************************************************************************************************)
A_TransportState();

(**************************************************************************************************************
   Takeover state
***************************************************************************************************************)
A_TakeOverState();                                                                                                                                                                 

(**************************************************************************************************************
   Handover state
***************************************************************************************************************)
A_HandOverState();

(**************************************************************************************************************
   Brake
***************************************************************************************************************)
A_Brake();

(**************************************************************************************************************
   Jam auto reset
***************************************************************************************************************)
A_JamAutoReset();

(**************************************************************************************************************
   Short zone restart
***************************************************************************************************************)
A_ShortZoneRestart();

(**************************************************************************************************************
   Output mapping
***************************************************************************************************************)
A_OutputMapping();

ACTION A_Brake:
(**************************************************************************************
 * 	NAME		A_Brake
 * 	FUNCTION	Determines the braking zone
 **************************************************************************************)

// Calculate stopping by accelaration
// s = v^2/2a
IF Acceleration <> 0 THEN
	StoppingByAccelaretion := (CurrentSpeed * CurrentSpeed) / (2 * Acceleration);
ELSE
	StoppingByAccelaretion := 0;
END_IF

// If the TU is on the way to the occupied position
IF NOT ZoneData.TransportControlData.Occupied THEN
	// If the TU is within the zone
	IF fbTrackingLeadingEdge.Run AND
	   fbTrackingLeadingEdge.Displacement <= UINT_TO_DINT(TransportParam.ZoneLength) THEN	  
		IF ZoneData.TransportControlData.FastSpeedActive THEN
			// TU is over the braking point	
			IF fbTrackingLeadingEdge.Displacement >= UINT_TO_DINT(TransportParam.ZoneLength)
			   - TransportParam.ZoneEndLength
			   + TransportParam.StopDelayDistance
			   - StoppingDistance
			   - StoppingByAccelaretion THEN
				// Set flag TU within braking zone
				TU_WithinBrakingZone := TRUE;
			END_IF
		END_IF
	END_IF

// If no transport before occupied is active	
ELSIF ZoneData.TransportControlData.eTransportState <> E_TransportState.TAKEOVER AND
	ZoneData.TransportControlData.eTransportState <> E_TransportState.FEEDIN AND
    ZoneData.TransportControlData.eTransportState <> E_TransportState.SIMULTANEOUS THEN
	TU_WithinBrakingZone := FALSE;
END_IF
END_ACTION

ACTION A_HandOverState:
(**************************************************************************************
 * 	NAME		A_HandOverState
 * 	FUNCTION	Handover state
 **************************************************************************************)

// If the transport is aborted set the interface to idle
IF ZoneData.TransportControlData.eTransportState = E_TransportState.IDLE OR
   ZoneData.TransportControlData.eTransportState = E_TransportState.CLEARING THEN
	ZoneData.TransportControlData.eHandOverState := E_HandOverState.IDLE;
END_IF

// Restet transport data request
HandOverTrspDataReq := InitTrspDataReq;
 
CASE ZoneData.TransportControlData.eHandOverState OF
(*************************************************************************
  Idle
*************************************************************************)
	E_HandOverState.IDLE:

		DriveHandoverRun := FALSE;

		// Reset zone end length clear	
		fbZoneEndLengthClear(Run := FALSE);

		// Reset jam monitoring
		IF NOT ZoneData.TransportControlData.Occupied THEN
			// Reset jam monitoring
			fbTimeoutJam(Run := FALSE);
		END_IF
	
		// Zone is ready to handover
		IF Inputs.Enable.Transport AND Inputs.Enable.HandOver AND
		   Param.rOperationState.eState = E_PositionState.STARTED AND
		   ErrorData.ErrorType <> E_ErrorType.ERROR THEN
			// If next zone or function is available
			IF NextTransportData.eFunctionNumber <> E_FunctionNumber.F_BEGIN_FUNCTION OR
			   Param.reNextFunctionNumber <> E_FunctionNumber.F_BEGIN_FUNCTION THEN	
				IF (ZoneData.TransportControlData.eTransportState = E_TransportState.HANDOVER OR
				   ZoneData.TransportControlData.eTransportState = E_TransportState.MULTIZONE_OCCUPIED OR
				   ZoneData.TransportControlData.eTransportState = E_TransportState.MULTIZONE_STOP OR
				   ZoneData.TransportControlData.eTransportState = E_TransportState.MULTI_TU_OCCUPIED OR
				   (ZoneData.TransportControlData.eTransportState = E_TransportState.MULTI_TU AND
					ZoneData.TransportControlData.Occupied) OR 
				     (ZoneData.TransportControlData.eTransportState = E_TransportState.SIMULTANEOUS_OCCUPIED AND
					  PrevTransportData.rTransportControlData.eHandOverState = E_HandOverState.READY AND
					  (NOT Param.rSettings.EnableMFC OR TU_DataTable[ZoneData.TransportControlData.TU_DataIndex].DataSet.JobPresent)) OR
				    ZoneData.TransportControlData.eTransportState = E_TransportState.SIMULTANEOUS_STOP) AND 
					DriveReady THEN
					ZoneData.TransportControlData.eHandOverState := E_HandOverState.READY;
					// Update for this transport valid trasport parameter
					TransportParam := ZoneData.TransportControlData.TransportParam;				
				END_IF
			END_IF		
		END_IF

(*************************************************************************
  Ready
*************************************************************************)
	E_HandOverState.READY:

		DriveHandoverRun := FALSE;

		// Next position started takeover
		IF NextTransportData.rTransportControlData.eTakeOverState = E_TakeOverState.ACTIVE THEN
			DriveHandoverRun := TRUE;
			ZoneData.TransportControlData.eHandOverState := E_HandOverState.ACTIVE;

		ELSIF NOT Inputs.Enable.Transport OR NOT Inputs.Enable.HandOver OR
			  Param.rOperationState.eState <> E_PositionState.STARTED OR
			  ErrorData.ErrorType = E_ErrorType.ERROR OR
			  (NextTransportData.eFunctionNumber = E_FunctionNumber.F_BEGIN_FUNCTION AND
			   Param.reNextFunctionNumber = E_FunctionNumber.F_BEGIN_FUNCTION) OR
			  ZoneData.TransportControlData.eTransportState <> E_TransportState.HANDOVER AND
		      ZoneData.TransportControlData.eTransportState <> E_TransportState.MULTIZONE_OCCUPIED AND
			  ZoneData.TransportControlData.eTransportState <> E_TransportState.MULTIZONE AND
		      ZoneData.TransportControlData.eTransportState <> E_TransportState.MULTIZONE_STOP AND
			  ZoneData.TransportControlData.eTransportState <> E_TransportState.MULTI_TU_OCCUPIED AND
			  (ZoneData.TransportControlData.eTransportState <> E_TransportState.MULTI_TU OR NOT
			   ZoneData.TransportControlData.Occupied) AND
			   (ZoneData.TransportControlData.eTransportState <> E_TransportState.SIMULTANEOUS_OCCUPIED OR 
                PrevTransportData.rTransportControlData.eHandOverState <> E_HandOverState.READY OR
				Param.rSettings.EnableMFC AND NOT TU_DataTable[ZoneData.TransportControlData.TU_DataIndex].DataSet.JobPresent) AND
			  ZoneData.TransportControlData.eTransportState <> E_TransportState.SIMULTANEOUS AND
			    ZoneData.TransportControlData.eTransportState <> E_TransportState.SIMULTANEOUS_STOP THEN
			HandOverTrspDataReq.DeleteNextTransportData := TRUE;   
			DriveHandoverRun := FALSE;
			ZoneData.TransportControlData.eHandOverState := E_HandOverState.IDLE;
		END_IF

(*************************************************************************
  Active
*************************************************************************)
	E_HandOverState.ACTIVE:
		// Set drive on
		DriveHandoverRun := TRUE;

		// If the zone is free
		IF NOT ZoneOccupiedSignal THEN
			// Run zone end length clearing 
			fbZoneEndLengthClear(
				Run 				:= TRUE,
				EncoderValueInc 	:= EncoderValue,
				MaxEncoderValueInc 	:= MaxEncoderValue,
				RateIncPerMM		:= 1,
				SetPoint 			:= TransportParam.ZoneEndLength);
		END_IF

		// Stop handover
		IF NOT Inputs.Enable.Transport OR
			ErrorData.ErrorType = E_ErrorType.ERROR OR
			Param.rOperationState.eState = E_PositionState.STOPPED OR
			ZoneData.TransportControlData.eTransportState = E_TransportState.MULTIZONE_STOP OR
			ZoneData.TransportControlData.eTransportState = E_TransportState.MULTI_TU_STOP OR 
			NOT DriveReady THEN
			DriveHandoverRun := FALSE;
			ZoneData.TransportControlData.eHandOverState := E_HandOverState.STOP;		
		
		// Complete handover if the zone is no longer occupied and the zone end length is clear -> regular completion without MFC
		ELSIF NOT ZoneData.TransportControlData.Occupied AND fbZoneEndLengthClear.Q THEN
			fbZoneEndLengthClear(Run := FALSE);
			DriveHandoverRun := TRUE;
			ZoneData.TransportControlData.eHandOverState := E_HandOverState.COMPLETE;		
		
		// Next position stopped takeover
		ELSIF NextTransportData.rTransportControlData.eTakeOverState = E_TakeOverState.STOP THEN
			// Interrupt handover if the zone is occupied 						
			IF ZoneData.TransportControlData.Occupied THEN
				DriveHandoverRun := FALSE;
				ZoneData.TransportControlData.eHandOverState := E_HandOverState.INTERRUPTED;
			// Oterwise end handover because the TU can no more be stopped on the zone
            // and the zone is already able to takeover a new TU
			ELSE
				fbZoneEndLengthClear(Run := FALSE);
				DriveHandoverRun := TRUE;
				ZoneData.TransportControlData.eHandOverState := E_HandOverState.COMPLETE;		
			END_IF
			
		// Next position aborted the takeover or the link is broken
		ELSIF NextTransportData.rTransportControlData.eTakeOverState = E_TakeOverState.IDLE OR
			  NextTransportData.rTransportControlData.eTakeOverState = E_TakeOverState.UNDEFINED THEN
			IF ZoneData.TransportControlData.Occupied THEN
				IF Param.rSettings.EnableMultipleTU_Transition THEN
					ZoneData.TransportControlData.NumberOfPresentTUs:= ZoneData.TransportControlData.NumberOfPresentTUs + 1;
				ELSE
					ZoneData.TransportControlData.NumberOfPresentTUs:= 1;
				END_IF
			END_IF
			HandOverTrspDataReq.DeleteNextTransportData := TRUE;
			DriveHandoverRun := FALSE;
			ZoneData.TransportControlData.eHandOverState := E_HandOverState.IDLE;

		// End handover if next position completed the takeover -> regular end with MFC
		ELSIF NextTransportData.rTransportControlData.eTakeOverState = E_TakeOverState.COMPLETE THEN
			IF NOT Param.rSettings.EnableMFC THEN
				// debug message: '11-001-0095-01-1,  takeover complete before handover complete (multizone?),  occupied = false,  end length = 25'
				DebugMsg := '';
				DebugMsg := CONCAT(DebugMsg, F_AddDividerToSisString(Param.rSettings.ZoneName));
				DebugMsg := CONCAT(DebugMsg, ',  takeover complete before handover complete (multizone?)');
				DebugMsg := CONCAT(DebugMsg, DebugTextBlocks.OCCUPIED);
				DebugMsg := CONCAT(DebugMsg, BOOL_TO_STRING(ZoneData.TransportControlData.Occupied));
				DebugMsg := CONCAT(DebugMsg, DebugTextBlocks.ENDLENGTH);
				DebugMsg := CONCAT(DebugMsg, DINT_TO_STRING(fbZoneEndLengthClear.SetPoint - fbZoneEndLengthClear.Displacement));
				fbDebugMsg.M_SendErrorMsg(DebugMsg);
			END_IF

			HandOverTrspDataReq.DeleteNextTransportData := TRUE;
			DriveHandoverRun := FALSE;
			ZoneData.TransportControlData.eHandOverState := E_HandOverState.IDLE;

		// If not multizone transport is active
		ELSIF ZoneData.TransportControlData.eTransportState <> E_TransportState.MULTIZONE AND
              NextTransportData.rTransportControlData.eTransportState <> E_TransportState.MULTIZONE_STOP AND
              NOT Param.rSettings.EnableMFC AND
			  CurrentSpeed > 0 THEN
			
			// Jam monitoring
			fbTimeoutJam(
				Run 				:= ZoneOccupiedSignal,
				EncoderValueInc 	:= EncoderValue,
				MaxEncoderValueInc 	:= MaxEncoderValue,
				RateIncPerMM		:= 1,
				SetPoint			:= Param.rSettings.JamTriggerDistance);

			// If timeout jam			
			IF fbTimeoutJam.Q THEN
				// If not short zone restart (A_ShortZoneRestart)			
				IF NOT EnableShortZoneRestart THEN
					// Set error
					F_SetError(	
						ErrorType	:= E_ErrorType.ERROR,
						ErrorParam	:= '',
						ErrorMsg	:= E_ErrorConv.JAM_ERROR,
						ErrorData	:= ErrorData);
					
					fbTimeoutJam(Run := FALSE);
				END_IF

				// Stop handover
				DriveHandoverRun := FALSE;
				ZoneData.TransportControlData.eHandOverState := E_HandOverState.STOP;
			END_IF				
		END_IF

(*************************************************************************
  Stop
*************************************************************************)
	E_HandOverState.STOP:

		DriveHandoverRun := FALSE;

		// If the next position aborted the takeover or the link is broken,
		// cancel the started handover
		IF NextTransportData.rTransportControlData.eTakeOverState = E_TakeOverState.IDLE OR
		   NextTransportData.rTransportControlData.eTakeOverState = E_TakeOverState.UNDEFINED THEN
			HandOverTrspDataReq.DeleteNextTransportData := TRUE;
			DriveHandoverRun := FALSE;
			ZoneData.TransportControlData.eHandOverState := E_HandOverState.IDLE;

		// If transport is enabled and position is started
		ELSIF Inputs.Enable.Transport AND
		   Param.rOperationState.eState = E_PositionState.STARTED THEN
			// If no error is pending
			IF ErrorData.ErrorType <> E_ErrorType.ERROR AND DriveReady THEN
				// If the transport state the execution allows
				IF ZoneData.TransportControlData.eTransportState <> E_TransportState.MULTIZONE_STOP AND
				   ZoneData.TransportControlData.eTransportState <> E_TransportState.MULTI_TU_STOP THEN
					DriveHandoverRun := TRUE;
					ZoneData.TransportControlData.eHandOverState := E_HandOverState.ACTIVE;
				END_IF
			END_IF
		END_IF

(*************************************************************************
  Interrupted
*************************************************************************)
	E_HandOverState.INTERRUPTED:

		DriveHandoverRun := FALSE;

		// If the next position aborted the takeover or the link is broken,
		// cancel the started handover
		IF NextTransportData.rTransportControlData.eTakeOverState = E_TakeOverState.IDLE OR
		   NextTransportData.rTransportControlData.eTakeOverState = E_TakeOverState.UNDEFINED THEN
			HandOverTrspDataReq.DeleteNextTransportData := TRUE;
			DriveHandoverRun := FALSE;
			ZoneData.TransportControlData.eHandOverState := E_HandOverState.IDLE;

		// If the next position is active again
		ELSIF NextTransportData.rTransportControlData.eTakeOverState = E_TakeOverState.ACTIVE THEN
			DriveHandoverRun := TRUE;
			ZoneData.TransportControlData.eHandOverState := E_HandOverState.ACTIVE;
		END_IF
		
(*************************************************************************
  Complete
*************************************************************************)
	E_HandOverState.COMPLETE:

		DriveHandoverRun := TRUE;

		// Set drive on
		DriveHandoverRun := NextTransportData.rTransportControlData.eTakeOverState <> E_TakeOverState.STOP AND
                            ZoneData.TransportControlData.eTransportState <> E_TransportState.OCCUPIED;
		
		// No pending transfer -> change to idle
		IF NextTransportData.rTransportControlData.eTakeOverState = E_TakeOverState.COMPLETE OR
		   NextTransportData.rTransportControlData.eTakeOverState = E_TakeOverState.READY OR
		   NextTransportData.rTransportControlData.eTakeOverState = E_TakeOverState.IDLE OR
		   NextTransportData.rTransportControlData.eTakeOverState = E_TakeOverState.UNDEFINED THEN
			HandOverTrspDataReq.DeleteNextTransportData := TRUE;
			DriveHandoverRun := FALSE;
			ZoneData.TransportControlData.eHandOverState := E_HandOverState.IDLE;
		END_IF

(*************************************************************************
  State error
*************************************************************************)
ELSE
	// Set error
	F_SetError(	
		ErrorType	:= E_ErrorType.ERROR,
		ErrorParam	:= INT_TO_STRING(ZoneData.TransportControlData.eHandOverState),
		ErrorMsg	:= E_ErrorConv.SOFTWARE_ERROR,
		ErrorData	:= ErrorData);
END_CASE
END_ACTION

ACTION A_Init:
(**************************************************************************************
 * 	NAME		A_Init
 * 	FUNCTION	Initialize
 **************************************************************************************)

// When zone is not initialized or invalid inputs are available
IF NOT ZoneData.Init THEN
	// Reset internal variables
	ZoneData.TransportControlData.eTransportState := E_TransportState.IDLE;
	ZoneData.TransportControlData.eTakeOverState := E_TakeOverState.IDLE;
	ZoneData.TransportControlData.eHandOverState := E_HandOverState.IDLE;
	Init := FALSE;

	TransportTrspDataReq := InitTrspDataReq;
	TakeOverTrspDataReq := InitTrspDataReq;
	HandOverTrspDataReq := InitTrspDataReq;

	EnableFastSpeed := TRUE;
	ErrorData.ResetError := TRUE;
	Outputs.DriveRun   				 := FALSE;
	Outputs.DriveTakeoverRun		 := FALSE;
	Outputs.DriveHandoverRun		 := FALSE;
	Outputs.RequestPrevTransportData := FALSE;
	Outputs.RequestNextTransportData := FALSE;
	Outputs.DeletePrevTransportData	 := FALSE;
	Outputs.DeleteNextTransportData  := FALSE;
	Outputs.DistanceToZoneEnd		 := 0;

